# B&R Automation Studio project MotionTestBenchMaster (part 7)

#### FB_ITC.st
```iecst
FUNCTION_BLOCK FB_HMI_ITC_DigitalBool
	VAR_ProgressiveId := INT_TO_UINT(FC_ReminderShift(UINT_TO_INT(Index), 16, 0));

	IF IN_ReadOnly OR IN_HMIAutoForce THEN
		VAR_Auto	:= TRUE;
		VAR_Man		:= FALSE;
	END_IF

	IF IN_IOType THEN
		ITC_IO 	:= SEL(VAR_Auto, VAR_Man, ITC);
	ELSE
		ITC 	:= SEL(VAR_Auto, VAR_Man, ITC_IO);
	END_IF

	IF VAR_OldPage <> HMI_Page.PageNum THEN
		VAR_PageSwitch	:= TRUE;
	END_IF

	IF (Index = (VAR_ProgressiveId + 16 * HMI_Page.PageNum)) AND IN_Visibility THEN
		IF VAR_PageSwitch THEN
			IF IN_IOType THEN
				HMI_Data.DigitalOut[VAR_ProgressiveId].Auto	:= VAR_Auto;
				HMI_Data.DigitalOut[VAR_ProgressiveId].Man	:= VAR_Man;
			ELSE
				HMI_Data.DigitalIn[VAR_ProgressiveId].Auto	:= VAR_Auto;
				HMI_Data.DigitalIn[VAR_ProgressiveId].Man	:= VAR_Man;
			END_IF
			VAR_PageSwitch	:= FALSE;
		END_IF

		IF IN_IOType THEN
			HMI_Data.DigitalOut[VAR_ProgressiveId].Visibility	:= IN_Visibility;
			HMI_Data.DigitalOut[VAR_ProgressiveId].Enable		:= NOT IN_ReadOnly AND NOT IN_HMIAutoForce;
			HMI_Data.DigitalOut[VAR_ProgressiveId].LampState	:= ITC_IO;
			HMI_Data.DigitalOut[VAR_ProgressiveId].Wait			:= IN_Wait;
			HMI_Data.DigitalOut[VAR_ProgressiveId].Alarm		:= IN_Alarm;
			HMI_Data.DigitalOut[VAR_ProgressiveId].Description	:= IN_Description;

			IF EDGEPOS(HMI_Data.DigitalOut[VAR_ProgressiveId].Auto) THEN
				HMI_Data.DigitalOut[VAR_ProgressiveId].Man := FALSE;
			ELSIF EDGEPOS(HMI_Data.DigitalOut[VAR_ProgressiveId].Man) THEN
				HMI_Data.DigitalOut[VAR_ProgressiveId].Auto := FALSE;
			END_IF

			IF IN_ReadOnly OR IN_HMIAutoForce THEN
				HMI_Data.DigitalOut[VAR_ProgressiveId].Auto	:= TRUE;
				HMI_Data.DigitalOut[VAR_ProgressiveId].Man	:= FALSE;
			END_IF

			VAR_Auto	:= HMI_Data.DigitalOut[VAR_ProgressiveId].Auto;
			VAR_Man		:= HMI_Data.DigitalOut[VAR_ProgressiveId].Man;
		ELSE
			HMI_Data.DigitalIn[VAR_ProgressiveId].Visibility	:= IN_Visibility;
			HMI_Data.DigitalIn[VAR_ProgressiveId].Enable		:= NOT IN_ReadOnly AND NOT IN_HMIAutoForce;
			HMI_Data.DigitalIn[VAR_ProgressiveId].LampState 	:= ITC;
			HMI_Data.DigitalIn[VAR_ProgressiveId].Wait			:= IN_Wait;
			HMI_Data.DigitalIn[VAR_ProgressiveId].Alarm			:= IN_Alarm;
			HMI_Data.DigitalIn[VAR_ProgressiveId].Description	:= IN_Description;

			IF EDGEPOS(HMI_Data.DigitalIn[VAR_ProgressiveId].Auto) THEN
				HMI_Data.DigitalIn[VAR_ProgressiveId].Man := FALSE;
			ELSIF EDGEPOS(HMI_Data.DigitalIn[VAR_ProgressiveId].Man) THEN
				HMI_Data.DigitalIn[VAR_ProgressiveId].Auto := FALSE;
			END_IF

			IF IN_ReadOnly OR IN_HMIAutoForce THEN
				HMI_Data.DigitalIn[VAR_ProgressiveId].Auto	:= TRUE;
				HMI_Data.DigitalIn[VAR_ProgressiveId].Man	:= FALSE;
			END_IF

			VAR_Auto	:= HMI_Data.DigitalIn[VAR_ProgressiveId].Auto;
			VAR_Man		:= HMI_Data.DigitalIn[VAR_ProgressiveId].Man;
		END_IF
	ELSIF (Index < (VAR_ProgressiveId + 16 * HMI_Page.PageNum)) THEN
		IF IN_IOType THEN
			HMI_Data.DigitalOut[VAR_ProgressiveId].Visibility	:= FALSE;
		ELSE
			HMI_Data.DigitalIn[VAR_ProgressiveId].Visibility	:= FALSE;
		END_IF
	END_IF

	VAR_OldPage := HMI_Page.PageNum;

	HMI_Data.ManActive	:= NOT VAR_Auto OR HMI_Data.ManActive;

	IF (Index > (16 + 16 * HMI_Page.PageNum)) AND IN_Visibility THEN
		HMI_Data.PageUp.Enable := TRUE;
	END_IF

	IF HMI_Page.PageNum <> 0 THEN
		HMI_Data.PageDown.Enable := TRUE;
	END_IF

	OUT_Man			:= NOT VAR_Auto;
	OUT_ManValue	:= VAR_Man;
	Index			:= Index + 1;
END_FUNCTION_BLOCK

FUNCTION_BLOCK FB_HMI_ITC_DigitalByte
	VAR_ProgressiveId := INT_TO_UINT(FC_ReminderShift(UINT_TO_INT(Index), 16, 0));

	IF IN_ReadOnly OR IN_HMIAutoForce THEN
		VAR_Auto	:= TRUE;
		VAR_Man		:= FALSE;
	END_IF

	IF IN_IOType THEN
		FOR VAR_BitIndex := 0 TO 7 DO
			IF VAR_BitIndex = INT_TO_USINT(IN_BitNumber) THEN
				IF NOT VAR_Auto THEN
					VAR_BitArray[VAR_BitIndex] := VAR_Man;
				ELSE
					VAR_BitArray[VAR_BitIndex] := ITC;
				END_IF
			ELSE
				VAR_BitArray[VAR_BitIndex] := (ITC_IO AND REAL_TO_BYTE(pow(2, VAR_BitIndex))) <> 0;
			END_IF
		END_FOR

		ITC_IO	:= 0;

		FOR VAR_BitIndex := 0 TO 7 DO
			ITC_IO	:= ITC_IO OR UINT_TO_BYTE(((REAL_TO_UINT(pow(2, VAR_BitIndex))) * VAR_BitArray[VAR_BitIndex]));
		END_FOR
	ELSE
		IF NOT VAR_Auto THEN
			ITC		:= VAR_Man;
		ELSE
			ITC		:= (ITC_IO AND REAL_TO_BYTE(pow(2, IN_BitNumber))) <> 0;
		END_IF
	END_IF

	IF VAR_OldPage <> HMI_Page.PageNum THEN
		VAR_PageSwitch	:= TRUE;
	END_IF

	IF (Index = (VAR_ProgressiveId + 16 * HMI_Page.PageNum)) AND IN_Visibility THEN
		IF VAR_PageSwitch THEN
			IF IN_IOType THEN
				HMI_Data.DigitalOut[VAR_ProgressiveId].Auto	:= VAR_Auto;
				HMI_Data.DigitalOut[VAR_ProgressiveId].Man	:= VAR_Man;
			ELSE
				HMI_Data.DigitalIn[VAR_ProgressiveId].Auto	:= VAR_Auto;
				HMI_Data.DigitalIn[VAR_ProgressiveId].Man	:= VAR_Man;
			END_IF
			VAR_PageSwitch	:= FALSE;
		END_IF

		IF IN_IOType THEN
			HMI_Data.DigitalOut[VAR_ProgressiveId].Visibility	:= IN_Visibility;
			HMI_Data.DigitalOut[VAR_ProgressiveId].Enable		:= NOT IN_ReadOnly AND NOT IN_HMIAutoForce;
			HMI_Data.DigitalOut[VAR_ProgressiveId].LampState	:= (ITC_IO AND REAL_TO_BYTE(pow(2, IN_BitNumber))) <> 0;
			HMI_Data.DigitalOut[VAR_ProgressiveId].Wait			:= IN_Wait;
			HMI_Data.DigitalOut[VAR_ProgressiveId].Alarm		:= IN_Alarm;
			HMI_Data.DigitalOut[VAR_ProgressiveId].Description	:= IN_Description;

			IF EDGEPOS(HMI_Data.DigitalOut[VAR_ProgressiveId].Auto) THEN
				HMI_Data.DigitalOut[VAR_ProgressiveId].Man := FALSE;
			ELSIF EDGEPOS(HMI_Data.DigitalOut[VAR_ProgressiveId].Man) THEN
				HMI_Data.DigitalOut[VAR_ProgressiveId].Auto := FALSE;
			END_IF

			IF IN_ReadOnly OR IN_HMIAutoForce THEN
				HMI_Data.DigitalOut[VAR_ProgressiveId].Auto	:= TRUE;
				HMI_Data.DigitalOut[VAR_ProgressiveId].Man	:= FALSE;
			END_IF

			VAR_Auto	:= HMI_Data.DigitalOut[VAR_ProgressiveId].Auto;
			VAR_Man		:= HMI_Data.DigitalOut[VAR_ProgressiveId].Man;
		ELSE
			HMI_Data.DigitalIn[VAR_ProgressiveId].Visibility	:= IN_Visibility;
			HMI_Data.DigitalIn[VAR_ProgressiveId].Enable		:= NOT IN_ReadOnly AND NOT IN_HMIAutoForce;
			HMI_Data.DigitalIn[VAR_ProgressiveId].LampState 	:= ITC;
			HMI_Data.DigitalIn[VAR_ProgressiveId].Wait			:= IN_Wait;
			HMI_Data.DigitalIn[VAR_ProgressiveId].Alarm			:= IN_Alarm;
			HMI_Data.DigitalIn[VAR_ProgressiveId].Description	:= IN_Description;

			IF EDGEPOS(HMI_Data.DigitalIn[VAR_ProgressiveId].Auto) THEN
				HMI_Data.DigitalIn[VAR_ProgressiveId].Man := FALSE;
			ELSIF EDGEPOS(HMI_Data.DigitalIn[VAR_ProgressiveId].Man) THEN
				HMI_Data.DigitalIn[VAR_ProgressiveId].Auto := FALSE;
			END_IF

			IF IN_ReadOnly OR IN_HMIAutoForce THEN
				HMI_Data.DigitalIn[VAR_ProgressiveId].Auto	:= TRUE;
				HMI_Data.DigitalIn[VAR_ProgressiveId].Man	:= FALSE;
			END_IF

			VAR_Auto	:= HMI_Data.DigitalIn[VAR_ProgressiveId].Auto;
			VAR_Man		:= HMI_Data.DigitalIn[VAR_ProgressiveId].Man;
		END_IF
	ELSIF (Index < (VAR_ProgressiveId + 16 * HMI_Page.PageNum)) THEN
		IF IN_IOType THEN
			HMI_Data.DigitalOut[VAR_ProgressiveId].Visibility	:= FALSE;
		ELSE
			HMI_Data.DigitalIn[VAR_ProgressiveId].Visibility	:= FALSE;
		END_IF
	END_IF

	VAR_OldPage := HMI_Page.PageNum;

	HMI_Data.ManActive	:= NOT VAR_Auto OR HMI_Data.ManActive;

	IF (Index > (16 + 16 * HMI_Page.PageNum)) AND IN_Visibility THEN
		HMI_Data.PageUp.Enable := TRUE;
	END_IF

	IF HMI_Page.PageNum <> 0 THEN
		HMI_Data.PageDown.Enable := TRUE;
	END_IF

	OUT_Man			:= NOT VAR_Auto;
	OUT_ManValue	:= VAR_Man;
	Index			:= Index + 1;
END_FUNCTION_BLOCK

FUNCTION_BLOCK FB_HMI_ITC_DigitalUsint
	VAR_ProgressiveId := INT_TO_UINT(FC_ReminderShift(UINT_TO_INT(Index), 16, 0));

	IF IN_ReadOnly OR IN_HMIAutoForce THEN
		VAR_Auto	:= TRUE;
		VAR_Man		:= FALSE;
	END_IF

	IF IN_IOType THEN
		FOR VAR_BitIndex := 0 TO 7 DO
			IF VAR_BitIndex = INT_TO_USINT(IN_BitNumber) THEN
				IF NOT VAR_Auto THEN
					VAR_BitArray[VAR_BitIndex] := VAR_Man;
				ELSE
					VAR_BitArray[VAR_BitIndex] := ITC;
				END_IF
			ELSE
				VAR_BitArray[VAR_BitIndex] := (ITC_IO AND REAL_TO_USINT(pow(2, VAR_BitIndex))) <> 0;
			END_IF
		END_FOR

		ITC_IO	:= 0;

		FOR VAR_BitIndex := 0 TO 7 DO
			ITC_IO	:= ITC_IO OR UINT_TO_USINT(((REAL_TO_UINT(pow(2, VAR_BitIndex))) * VAR_BitArray[VAR_BitIndex]));
		END_FOR
	ELSE
		IF NOT VAR_Auto THEN
			ITC		:= VAR_Man;
		ELSE
			ITC		:= (ITC_IO AND REAL_TO_USINT(pow(2, IN_BitNumber))) <> 0;
		END_IF
	END_IF

	IF VAR_OldPage <> HMI_Page.PageNum THEN
		VAR_PageSwitch	:= TRUE;
	END_IF

	IF (Index = (VAR_ProgressiveId + 16 * HMI_Page.PageNum(*VAR_OldPage*))) AND IN_Visibility THEN
		IF VAR_PageSwitch THEN
			IF IN_IOType THEN
				HMI_Data.DigitalOut[VAR_ProgressiveId].Auto	:= VAR_Auto;
				HMI_Data.DigitalOut[VAR_ProgressiveId].Man	:= VAR_Man;
			ELSE
				HMI_Data.DigitalIn[VAR_ProgressiveId].Auto	:= VAR_Auto;
				HMI_Data.DigitalIn[VAR_ProgressiveId].Man	:= VAR_Man;
			END_IF
			VAR_PageSwitch	:= FALSE;
		END_IF

		IF IN_IOType THEN
			HMI_Data.DigitalOut[VAR_ProgressiveId].Visibility	:= IN_Visibility;
			HMI_Data.DigitalOut[VAR_ProgressiveId].Enable		:= NOT IN_ReadOnly AND NOT IN_HMIAutoForce;
			HMI_Data.DigitalOut[VAR_ProgressiveId].LampState	:= (ITC_IO AND REAL_TO_USINT(pow(2, IN_BitNumber))) <> 0;
			HMI_Data.DigitalOut[VAR_ProgressiveId].Wait			:= IN_Wait;
			HMI_Data.DigitalOut[VAR_ProgressiveId].Alarm		:= IN_Alarm;
			HMI_Data.DigitalOut[VAR_ProgressiveId].Description	:= IN_Description;

			IF EDGEPOS(HMI_Data.DigitalOut[VAR_ProgressiveId].Auto) THEN
				HMI_Data.DigitalOut[VAR_ProgressiveId].Man := FALSE;
				VAR_Man		:= FALSE;
			ELSIF EDGEPOS(HMI_Data.DigitalOut[VAR_ProgressiveId].Man) THEN
				HMI_Data.DigitalOut[VAR_ProgressiveId].Auto := FALSE;
				VAR_Auto	:= FALSE;
			END_IF

			IF IN_ReadOnly OR IN_HMIAutoForce THEN
				HMI_Data.DigitalOut[VAR_ProgressiveId].Auto	:= TRUE;
				HMI_Data.DigitalOut[VAR_ProgressiveId].Man	:= FALSE;
			END_IF

			VAR_Auto	:= HMI_Data.DigitalOut[VAR_ProgressiveId].Auto;
			VAR_Man		:= HMI_Data.DigitalOut[VAR_ProgressiveId].Man;
		ELSE
			HMI_Data.DigitalIn[VAR_ProgressiveId].Visibility	:= IN_Visibility;
			HMI_Data.DigitalIn[VAR_ProgressiveId].Enable		:= NOT IN_ReadOnly AND NOT IN_HMIAutoForce;
			HMI_Data.DigitalIn[VAR_ProgressiveId].LampState 	:= ITC;
			HMI_Data.DigitalIn[VAR_ProgressiveId].Wait			:= IN_Wait;
			HMI_Data.DigitalIn[VAR_ProgressiveId].Alarm			:= IN_Alarm;
			HMI_Data.DigitalIn[VAR_ProgressiveId].Description	:= IN_Description;

			IF EDGEPOS(HMI_Data.DigitalIn[VAR_ProgressiveId].Auto) THEN
				HMI_Data.DigitalIn[VAR_ProgressiveId].Man := FALSE;
			ELSIF EDGEPOS(HMI_Data.DigitalIn[VAR_ProgressiveId].Man) THEN
				HMI_Data.DigitalIn[VAR_ProgressiveId].Auto := FALSE;
			END_IF

			IF IN_ReadOnly OR IN_HMIAutoForce THEN
				HMI_Data.DigitalIn[VAR_ProgressiveId].Auto	:= TRUE;
				HMI_Data.DigitalIn[VAR_ProgressiveId].Man	:= FALSE;
			END_IF

			VAR_Auto	:= HMI_Data.DigitalIn[VAR_ProgressiveId].Auto;
			VAR_Man		:= HMI_Data.DigitalIn[VAR_ProgressiveId].Man;
		END_IF
	ELSIF (Index < (VAR_ProgressiveId + 16 * HMI_Page.PageNum(*VAR_OldPage*))) THEN
		IF IN_IOType THEN
			HMI_Data.DigitalOut[VAR_ProgressiveId].Visibility	:= FALSE;
		ELSE
			HMI_Data.DigitalIn[VAR_ProgressiveId].Visibility	:= FALSE;
		END_IF
	END_IF

	VAR_OldPage := HMI_Page.PageNum;

	HMI_Data.ManActive	:= NOT VAR_Auto OR HMI_Data.ManActive;

	IF (Index > (16 + 16 * HMI_Page.PageNum)) AND IN_Visibility THEN
		HMI_Data.PageUp.Enable := TRUE;
	END_IF

	IF HMI_Page.PageNum <> 0 THEN
		HMI_Data.PageDown.Enable := TRUE;
	END_IF

	OUT_Man			:= NOT VAR_Auto;
	OUT_ManValue	:= VAR_Man;
	Index			:= Index + 1;
END_FUNCTION_BLOCK

FUNCTION_BLOCK FB_HMI_ITC_DigitalInt
	VAR_ProgressiveId := INT_TO_UINT(FC_ReminderShift(UINT_TO_INT(Index), 16, 0));

	IF IN_ReadOnly OR IN_HMIAutoForce THEN
		VAR_Auto	:= TRUE;
		VAR_Man		:= FALSE;
	END_IF

	IF IN_IOType THEN
		FOR VAR_BitIndex := 0 TO 15 DO
			IF VAR_BitIndex = INT_TO_USINT(IN_BitNumber) THEN
				IF NOT VAR_Auto THEN
					VAR_BitArray[VAR_BitIndex] := VAR_Man;
				ELSE
					VAR_BitArray[VAR_BitIndex] := ITC;
				END_IF
			ELSE
				VAR_BitArray[VAR_BitIndex] := (ITC_IO AND REAL_TO_INT(pow(2, VAR_BitIndex))) <> 0;
			END_IF
		END_FOR

		ITC_IO	:= 0;

		FOR VAR_BitIndex := 0 TO 15 DO
			ITC_IO	:= ITC_IO OR UINT_TO_INT(((REAL_TO_UINT(pow(2, VAR_BitIndex))) * VAR_BitArray[VAR_BitIndex]));
		END_FOR
	ELSE
		IF NOT VAR_Auto THEN
			ITC		:= VAR_Man;
		ELSE
			ITC		:= (ITC_IO AND REAL_TO_INT(pow(2, IN_BitNumber))) <> 0;
		END_IF
	END_IF

	IF VAR_OldPage <> HMI_Page.PageNum THEN
		VAR_PageSwitch	:= TRUE;
	END_IF

	IF (Index = (VAR_ProgressiveId + 16 * HMI_Page.PageNum)) AND IN_Visibility THEN
		IF VAR_PageSwitch THEN
			IF IN_IOType THEN
				HMI_Data.DigitalOut[VAR_ProgressiveId].Auto	:= VAR_Auto;
				HMI_Data.DigitalOut[VAR_ProgressiveId].Man	:= VAR_Man;
			ELSE
				HMI_Data.DigitalIn[VAR_ProgressiveId].Auto	:= VAR_Auto;
				HMI_Data.DigitalIn[VAR_ProgressiveId].Man	:= VAR_Man;
			END_IF
			VAR_PageSwitch	:= FALSE;
		END_IF

		IF IN_IOType THEN
			HMI_Data.DigitalOut[VAR_ProgressiveId].Visibility	:= IN_Visibility;
			HMI_Data.DigitalOut[VAR_ProgressiveId].Enable		:= NOT IN_ReadOnly AND NOT IN_HMIAutoForce;
			HMI_Data.DigitalOut[VAR_ProgressiveId].LampState	:= (ITC_IO AND REAL_TO_INT(pow(2, IN_BitNumber))) <> 0;
			HMI_Data.DigitalOut[VAR_ProgressiveId].Wait			:= IN_Wait;
			HMI_Data.DigitalOut[VAR_ProgressiveId].Alarm		:= IN_Alarm;
			HMI_Data.DigitalOut[VAR_ProgressiveId].Description	:= IN_Description;

			IF EDGEPOS(HMI_Data.DigitalOut[VAR_ProgressiveId].Auto) THEN
				HMI_Data.DigitalOut[VAR_ProgressiveId].Man := FALSE;
			ELSIF EDGEPOS(HMI_Data.DigitalOut[VAR_ProgressiveId].Man) THEN
				HMI_Data.DigitalOut[VAR_ProgressiveId].Auto := FALSE;
			END_IF

			VAR_Auto	:= HMI_Data.DigitalOut[VAR_ProgressiveId].Auto;
			VAR_Man		:= HMI_Data.DigitalOut[VAR_ProgressiveId].Man;
		ELSE
			HMI_Data.DigitalIn[VAR_ProgressiveId].Visibility	:= IN_Visibility;
			HMI_Data.DigitalIn[VAR_ProgressiveId].Enable		:= NOT IN_ReadOnly AND NOT IN_HMIAutoForce;
			HMI_Data.DigitalIn[VAR_ProgressiveId].LampState 	:= ITC;
			HMI_Data.DigitalIn[VAR_ProgressiveId].Wait			:= IN_Wait;
			HMI_Data.DigitalIn[VAR_ProgressiveId].Alarm			:= IN_Alarm;
			HMI_Data.DigitalIn[VAR_ProgressiveId].Description	:= IN_Description;

			IF EDGEPOS(HMI_Data.DigitalIn[VAR_ProgressiveId].Auto) THEN
				HMI_Data.DigitalIn[VAR_ProgressiveId].Man := FALSE;
			ELSIF EDGEPOS(HMI_Data.DigitalIn[VAR_ProgressiveId].Man) THEN
				HMI_Data.DigitalIn[VAR_ProgressiveId].Auto := FALSE;
			END_IF

			VAR_Auto	:= HMI_Data.DigitalIn[VAR_ProgressiveId].Auto;
			VAR_Man		:= HMI_Data.DigitalIn[VAR_ProgressiveId].Man;
		END_IF
	ELSIF (Index < (VAR_ProgressiveId + 16 * HMI_Page.PageNum)) THEN
		IF IN_IOType THEN
			HMI_Data.DigitalOut[VAR_ProgressiveId].Visibility	:= FALSE;
		ELSE
			HMI_Data.DigitalIn[VAR_ProgressiveId].Visibility	:= FALSE;
		END_IF
	END_IF

	VAR_OldPage := HMI_Page.PageNum;

	HMI_Data.ManActive	:= NOT VAR_Auto OR HMI_Data.ManActive;

	IF (Index > (16 + 16 * HMI_Page.PageNum)) AND IN_Visibility THEN
		HMI_Data.PageUp.Enable := TRUE;
	END_IF

	IF HMI_Page.PageNum <> 0 THEN
		HMI_Data.PageDown.Enable := TRUE;
	END_IF

	OUT_Man			:= NOT VAR_Auto;
	OUT_ManValue	:= VAR_Man;
	Index			:= Index + 1;
END_FUNCTION_BLOCK

FUNCTION_BLOCK FB_HMI_ITC_AnalogByte
	VAR_ProgressiveId := INT_TO_UINT(FC_ReminderShift(UINT_TO_INT(Index), 4, 0));

	IF IN_ReadOnly OR IN_HMIAutoForce THEN
		VAR_Man		:= FALSE;
	END_IF

	IF IN_IOType THEN
		ITC_IO 		:= SEL(VAR_Man, ITC, VAR_ManValue);
	ELSE
		ITC 		:= SEL(VAR_Man, ITC_IO, VAR_ManValue);
	END_IF

	IF VAR_OldPage <> HMI_Page.PageNum THEN
		VAR_PageSwitch	:= TRUE;
	END_IF

	IF (Index = (VAR_ProgressiveId + 4 * HMI_Page.PageNum)) AND IN_Visibility THEN
		IF VAR_PageSwitch THEN
			IF IN_IOType THEN
				HMI_Data.AnalogOut[VAR_ProgressiveId].Man		:= VAR_Man;
				HMI_Data.AnalogOut[VAR_ProgressiveId].PV_Man	:= BYTE_TO_REAL(VAR_ManValue);
			ELSE
				HMI_Data.AnalogIn[VAR_ProgressiveId].Man		:= VAR_Man;
				HMI_Data.AnalogIn[VAR_ProgressiveId].PV_Man		:= BYTE_TO_REAL(VAR_ManValue);
			END_IF
			VAR_PageSwitch	:= FALSE;
		END_IF

		IF IN_IOType THEN
			HMI_Data.AnalogOut[VAR_ProgressiveId].Visibility	:= IN_Visibility;
			HMI_Data.AnalogOut[VAR_ProgressiveId].Enable		:= NOT IN_ReadOnly AND NOT IN_HMIAutoForce;
			HMI_Data.AnalogOut[VAR_ProgressiveId].PV			:= BYTE_TO_REAL(ITC_IO);
			HMI_Data.AnalogOut[VAR_ProgressiveId].Wait			:= IN_Wait;
			HMI_Data.AnalogOut[VAR_ProgressiveId].Description	:= IN_Description;
			HMI_Data.AnalogOut[VAR_ProgressiveId].Unit			:= IN_Unit;
			HMI_Data.AnalogOut[VAR_ProgressiveId].MaxValue		:= IN_MaxValue;
			HMI_Data.AnalogOut[VAR_ProgressiveId].MinValue		:= IN_MinValue;

			VAR_Man			:= HMI_Data.AnalogOut[VAR_ProgressiveId].Man;
			VAR_ManValue	:= REAL_TO_BYTE(HMI_Data.AnalogOut[VAR_ProgressiveId].PV_Man);
		ELSE
			HMI_Data.AnalogIn[VAR_ProgressiveId].Visibility		:= IN_Visibility;
			HMI_Data.AnalogIn[VAR_ProgressiveId].Enable			:= NOT IN_ReadOnly AND NOT IN_HMIAutoForce;
			HMI_Data.AnalogIn[VAR_ProgressiveId].PV				:= BYTE_TO_REAL(ITC);
			HMI_Data.AnalogIn[VAR_ProgressiveId].Wait			:= IN_Wait;
			HMI_Data.AnalogIn[VAR_ProgressiveId].Description	:= IN_Description;
			HMI_Data.AnalogIn[VAR_ProgressiveId].Unit			:= IN_Unit;
			HMI_Data.AnalogIn[VAR_ProgressiveId].MaxValue		:= IN_MaxValue;
			HMI_Data.AnalogIn[VAR_ProgressiveId].MinValue		:= IN_MinValue;

			VAR_Man			:= HMI_Data.AnalogIn[VAR_ProgressiveId].Man;
			VAR_ManValue	:= REAL_TO_BYTE(HMI_Data.AnalogIn[VAR_ProgressiveId].PV_Man);
		END_IF
	ELSIF (Index < (VAR_ProgressiveId + 4 * HMI_Page.PageNum)) THEN
		IF IN_IOType THEN
			HMI_Data.AnalogOut[VAR_ProgressiveId].Visibility	:= FALSE;
		ELSE
			HMI_Data.AnalogIn[VAR_ProgressiveId].Visibility		:= FALSE;
		END_IF
	END_IF

	VAR_OldPage := HMI_Page.PageNum;

	HMI_Data.ManActive	:= VAR_Man OR HMI_Data.ManActive;

	IF (Index > (4 + 4 * HMI_Page.PageNum)) AND IN_Visibility THEN
		HMI_Data.PageUp.Enable := TRUE;
	END_IF

	IF HMI_Page.PageNum <> 0 THEN
		HMI_Data.PageDown.Enable := TRUE;
	END_IF

	OUT_Man			:= VAR_Man;
	OUT_ManValue	:= VAR_ManValue;
	Index			:= Index + 1;
END_FUNCTION_BLOCK

FUNCTION_BLOCK FB_HMI_ITC_AnalogUsint
	VAR_ProgressiveId := INT_TO_UINT(FC_ReminderShift(UINT_TO_INT(Index), 4, 0));

	IF IN_ReadOnly OR IN_HMIAutoForce THEN
		VAR_Man		:= FALSE;
	END_IF

	IF IN_IOType THEN
		ITC_IO 		:= SEL(VAR_Man, ITC, VAR_ManValue);
	ELSE
		ITC 		:= SEL(VAR_Man, ITC_IO, VAR_ManValue);
	END_IF

	IF VAR_OldPage <> HMI_Page.PageNum THEN
		VAR_PageSwitch	:= TRUE;
	END_IF

	IF (Index = (VAR_ProgressiveId + 4 * HMI_Page.PageNum)) AND IN_Visibility THEN
		IF VAR_PageSwitch THEN
			IF IN_IOType THEN
				HMI_Data.AnalogOut[VAR_ProgressiveId].Man		:= VAR_Man;
				HMI_Data.AnalogOut[VAR_ProgressiveId].PV_Man	:= USINT_TO_REAL(VAR_ManValue);
			ELSE
				HMI_Data.AnalogIn[VAR_ProgressiveId].Man		:= VAR_Man;
				HMI_Data.AnalogIn[VAR_ProgressiveId].PV_Man		:= USINT_TO_REAL(VAR_ManValue);
			END_IF
			VAR_PageSwitch	:= FALSE;
		END_IF

		IF IN_IOType THEN
			HMI_Data.AnalogOut[VAR_ProgressiveId].Visibility	:= IN_Visibility;
			HMI_Data.AnalogOut[VAR_ProgressiveId].Enable		:= NOT IN_ReadOnly AND NOT IN_HMIAutoForce;
			HMI_Data.AnalogOut[VAR_ProgressiveId].PV			:= USINT_TO_REAL(ITC_IO);
			HMI_Data.AnalogOut[VAR_ProgressiveId].Wait			:= IN_Wait;
			HMI_Data.AnalogOut[VAR_ProgressiveId].Description	:= IN_Description;
			HMI_Data.AnalogOut[VAR_ProgressiveId].Unit			:= IN_Unit;
			HMI_Data.AnalogOut[VAR_ProgressiveId].MaxValue		:= IN_MaxValue;
			HMI_Data.AnalogOut[VAR_ProgressiveId].MinValue		:= IN_MinValue;

			VAR_Man			:= HMI_Data.AnalogOut[VAR_ProgressiveId].Man;
			VAR_ManValue	:= REAL_TO_USINT(HMI_Data.AnalogOut[VAR_ProgressiveId].PV_Man);
		ELSE
			HMI_Data.AnalogIn[VAR_ProgressiveId].Visibility		:= IN_Visibility;
			HMI_Data.AnalogIn[VAR_ProgressiveId].Enable			:= NOT IN_ReadOnly AND NOT IN_HMIAutoForce;
			HMI_Data.AnalogIn[VAR_ProgressiveId].PV				:= USINT_TO_REAL(ITC);
			HMI_Data.AnalogIn[VAR_ProgressiveId].Wait			:= IN_Wait;
			HMI_Data.AnalogIn[VAR_ProgressiveId].Description	:= IN_Description;
			HMI_Data.AnalogIn[VAR_ProgressiveId].Unit			:= IN_Unit;
			HMI_Data.AnalogIn[VAR_ProgressiveId].MaxValue		:= IN_MaxValue;
			HMI_Data.AnalogIn[VAR_ProgressiveId].MinValue		:= IN_MinValue;

			VAR_Man			:= HMI_Data.AnalogIn[VAR_ProgressiveId].Man;
			VAR_ManValue	:= REAL_TO_USINT(HMI_Data.AnalogIn[VAR_ProgressiveId].PV_Man);
		END_IF
	ELSIF (Index < (VAR_ProgressiveId + 4 * HMI_Page.PageNum)) THEN
		IF IN_IOType THEN
			HMI_Data.AnalogOut[VAR_ProgressiveId].Visibility	:= FALSE;
		ELSE
			HMI_Data.AnalogIn[VAR_ProgressiveId].Visibility		:= FALSE;
		END_IF
	END_IF

	VAR_OldPage := HMI_Page.PageNum;

	HMI_Data.ManActive	:= VAR_Man OR HMI_Data.ManActive;

	IF (Index > (4 + 4 * HMI_Page.PageNum)) AND IN_Visibility THEN
		HMI_Data.PageUp.Enable := TRUE;
	END_IF

	IF HMI_Page.PageNum <> 0 THEN
		HMI_Data.PageDown.Enable := TRUE;
	END_IF

	OUT_Man			:= VAR_Man;
	OUT_ManValue	:= VAR_ManValue;
	Index			:= Index + 1;
END_FUNCTION_BLOCK

FUNCTION_BLOCK FB_HMI_ITC_AnalogInt
	VAR_ProgressiveId := INT_TO_UINT(FC_ReminderShift(UINT_TO_INT(Index), 4, 0));

	IF IN_ReadOnly OR IN_HMIAutoForce THEN
		VAR_Man		:= FALSE;
	END_IF

	IF IN_IOType THEN
		VAR_Value 	:= SEL(VAR_Man, ITC, VAR_ManValue);
		ITC_IO 		:= SEL(HMI_Data.ComSwap, VAR_Value, swapINT(VAR_Value));
	ELSE
		VAR_Value 	:= SEL(HMI_Data.ComSwap, ITC_IO, swapINT(ITC_IO));
		ITC 		:= SEL(VAR_Man, VAR_Value, VAR_ManValue);
	END_IF

	IF VAR_OldPage <> HMI_Page.PageNum THEN
		VAR_PageSwitch	:= TRUE;
	END_IF

	IF (Index = (VAR_ProgressiveId + 4 * HMI_Page.PageNum)) AND IN_Visibility THEN
		IF VAR_PageSwitch THEN
			IF IN_IOType THEN
				HMI_Data.AnalogOut[VAR_ProgressiveId].Man		:= VAR_Man;
				HMI_Data.AnalogOut[VAR_ProgressiveId].PV_Man	:= INT_TO_REAL(VAR_ManValue);
			ELSE
				HMI_Data.AnalogIn[VAR_ProgressiveId].Man		:= VAR_Man;
				HMI_Data.AnalogIn[VAR_ProgressiveId].PV_Man		:= INT_TO_REAL(VAR_ManValue);
			END_IF
			VAR_PageSwitch	:= FALSE;
		END_IF

		IF IN_IOType THEN
			HMI_Data.AnalogOut[VAR_ProgressiveId].Visibility	:= IN_Visibility;
			HMI_Data.AnalogOut[VAR_ProgressiveId].Enable		:= NOT IN_ReadOnly AND NOT IN_HMIAutoForce;
			HMI_Data.AnalogOut[VAR_ProgressiveId].PV			:= INT_TO_REAL(VAR_Value);
			HMI_Data.AnalogOut[VAR_ProgressiveId].Wait			:= IN_Wait;
			HMI_Data.AnalogOut[VAR_ProgressiveId].Description	:= IN_Description;
			HMI_Data.AnalogOut[VAR_ProgressiveId].Unit			:= IN_Unit;
			HMI_Data.AnalogOut[VAR_ProgressiveId].MaxValue		:= IN_MaxValue;
			HMI_Data.AnalogOut[VAR_ProgressiveId].MinValue		:= IN_MinValue;

			VAR_Man			:= HMI_Data.AnalogOut[VAR_ProgressiveId].Man;
			VAR_ManValue	:= REAL_TO_INT(HMI_Data.AnalogOut[VAR_ProgressiveId].PV_Man);
		ELSE
			HMI_Data.AnalogIn[VAR_ProgressiveId].Visibility		:= IN_Visibility;
			HMI_Data.AnalogIn[VAR_ProgressiveId].Enable			:= NOT IN_ReadOnly AND NOT IN_HMIAutoForce;
			HMI_Data.AnalogIn[VAR_ProgressiveId].PV				:= INT_TO_REAL(ITC);
			HMI_Data.AnalogIn[VAR_ProgressiveId].Wait			:= IN_Wait;
			HMI_Data.AnalogIn[VAR_ProgressiveId].Description	:= IN_Description;
			HMI_Data.AnalogIn[VAR_ProgressiveId].Unit			:= IN_Unit;
			HMI_Data.AnalogIn[VAR_ProgressiveId].MaxValue		:= IN_MaxValue;
			HMI_Data.AnalogIn[VAR_ProgressiveId].MinValue		:= IN_MinValue;

			VAR_Man			:= HMI_Data.AnalogIn[VAR_ProgressiveId].Man;
			VAR_ManValue	:= REAL_TO_INT(HMI_Data.AnalogIn[VAR_ProgressiveId].PV_Man);
		END_IF
	ELSIF (Index < (VAR_ProgressiveId + 4 * HMI_Page.PageNum)) THEN
		IF IN_IOType THEN
			HMI_Data.AnalogOut[VAR_ProgressiveId].Visibility	:= FALSE;
		ELSE
			HMI_Data.AnalogIn[VAR_ProgressiveId].Visibility		:= FALSE;
		END_IF
	END_IF

	VAR_OldPage := HMI_Page.PageNum;

	HMI_Data.ManActive	:= VAR_Man OR HMI_Data.ManActive;

	IF (Index > (4 + 4 * HMI_Page.PageNum)) AND IN_Visibility THEN
		HMI_Data.PageUp.Enable := TRUE;
	END_IF

	IF HMI_Page.PageNum <> 0 THEN
		HMI_Data.PageDown.Enable := TRUE;
	END_IF

	OUT_Man			:= VAR_Man;
	OUT_ManValue	:= VAR_ManValue;
	Index			:= Index + 1;
END_FUNCTION_BLOCK

FUNCTION_BLOCK FB_HMI_ITC_AnalogIntOverUsint
	VAR_ProgressiveId := INT_TO_UINT(FC_ReminderShift(UINT_TO_INT(Index), 4, 0));

	IF IN_ReadOnly OR IN_HMIAutoForce THEN
		VAR_Man		:= FALSE;
	END_IF

	IF IN_IOType THEN
		VAR_Value		:= SEL(VAR_Man, ITC, VAR_ManValue);
		VAR_RawValue	:= SEL(HMI_Data.ComSwap, VAR_Value, swapINT(VAR_Value));
		memcpy(ADR(ITC_IO), ADR(VAR_RawValue), SIZEOF(ITC));
	ELSE
		memcpy(ADR(VAR_RawValue), ADR(ITC_IO), SIZEOF(ITC));
		VAR_Value	:= SEL(HMI_Data.ComSwap, VAR_RawValue, swapINT(VAR_RawValue));
		ITC			:= SEL(VAR_Man, VAR_Value, VAR_ManValue);
	END_IF

	IF VAR_OldPage <> HMI_Page.PageNum THEN
		VAR_PageSwitch	:= TRUE;
	END_IF

	IF (Index = (VAR_ProgressiveId + 4 * HMI_Page.PageNum)) AND IN_Visibility THEN
		IF VAR_PageSwitch THEN
			IF IN_IOType THEN
				HMI_Data.AnalogOut[VAR_ProgressiveId].Man		:= VAR_Man;
				HMI_Data.AnalogOut[VAR_ProgressiveId].PV_Man	:= INT_TO_REAL(VAR_ManValue);
			ELSE
				HMI_Data.AnalogIn[VAR_ProgressiveId].Man		:= VAR_Man;
				HMI_Data.AnalogIn[VAR_ProgressiveId].PV_Man		:= INT_TO_REAL(VAR_ManValue);
			END_IF
			VAR_PageSwitch	:= FALSE;
		END_IF

		IF IN_IOType THEN
			HMI_Data.AnalogOut[VAR_ProgressiveId].Visibility	:= IN_Visibility;
			HMI_Data.AnalogOut[VAR_ProgressiveId].Enable		:= NOT IN_ReadOnly AND NOT IN_HMIAutoForce;
			HMI_Data.AnalogOut[VAR_ProgressiveId].PV			:= INT_TO_REAL(VAR_Value);
			HMI_Data.AnalogOut[VAR_ProgressiveId].Wait			:= IN_Wait;
			HMI_Data.AnalogOut[VAR_ProgressiveId].Description	:= IN_Description;
			HMI_Data.AnalogOut[VAR_ProgressiveId].Unit			:= IN_Unit;
			HMI_Data.AnalogOut[VAR_ProgressiveId].MaxValue		:= IN_MaxValue;
			HMI_Data.AnalogOut[VAR_ProgressiveId].MinValue		:= IN_MinValue;

			VAR_Man			:= HMI_Data.AnalogOut[VAR_ProgressiveId].Man;
			VAR_ManValue	:= REAL_TO_INT(HMI_Data.AnalogOut[VAR_ProgressiveId].PV_Man);
		ELSE
			HMI_Data.AnalogIn[VAR_ProgressiveId].Visibility		:= IN_Visibility;
			HMI_Data.AnalogIn[VAR_ProgressiveId].Enable			:= NOT IN_ReadOnly AND NOT IN_HMIAutoForce;
			HMI_Data.AnalogIn[VAR_ProgressiveId].PV				:= INT_TO_REAL(ITC);
			HMI_Data.AnalogIn[VAR_ProgressiveId].Wait			:= IN_Wait;
			HMI_Data.AnalogIn[VAR_ProgressiveId].Description	:= IN_Description;
			HMI_Data.AnalogIn[VAR_ProgressiveId].Unit			:= IN_Unit;
			HMI_Data.AnalogIn[VAR_ProgressiveId].MaxValue		:= IN_MaxValue;
			HMI_Data.AnalogIn[VAR_ProgressiveId].MinValue		:= IN_MinValue;

			VAR_Man			:= HMI_Data.AnalogIn[VAR_ProgressiveId].Man;
			VAR_ManValue	:= REAL_TO_INT(HMI_Data.AnalogIn[VAR_ProgressiveId].PV_Man);
		END_IF
	ELSIF (Index < (VAR_ProgressiveId + 4 * HMI_Page.PageNum)) THEN
		IF IN_IOType THEN
			HMI_Data.AnalogOut[VAR_ProgressiveId].Visibility	:= FALSE;
		ELSE
			HMI_Data.AnalogIn[VAR_ProgressiveId].Visibility		:= FALSE;
		END_IF
	END_IF

	VAR_OldPage := HMI_Page.PageNum;

	HMI_Data.ManActive	:= VAR_Man OR HMI_Data.ManActive;

	IF (Index > (4 + 4 * HMI_Page.PageNum)) AND IN_Visibility THEN
		HMI_Data.PageUp.Enable := TRUE;
	END_IF

	IF HMI_Page.PageNum <> 0 THEN
		HMI_Data.PageDown.Enable := TRUE;
	END_IF

	OUT_Man			:= VAR_Man;
	OUT_ManValue	:= VAR_ManValue;
	Index			:= Index + 1;
END_FUNCTION_BLOCK

FUNCTION_BLOCK FB_HMI_ITC_AnalogUintOverUsint
	VAR_ProgressiveId := INT_TO_UINT(FC_ReminderShift(UINT_TO_INT(Index), 4, 0));

	IF IN_ReadOnly OR IN_HMIAutoForce THEN
		VAR_Man		:= FALSE;
	END_IF

	IF IN_IOType THEN
		VAR_Value		:= SEL(VAR_Man, ITC, VAR_ManValue);
		VAR_RawValue	:= SEL(HMI_Data.ComSwap, VAR_Value, swapINT(VAR_Value));
		memcpy(ADR(ITC_IO), ADR(VAR_RawValue), SIZEOF(ITC));
	ELSE
		memcpy(ADR(VAR_RawValue), ADR(ITC_IO), SIZEOF(ITC));
		VAR_Value	:= SEL(HMI_Data.ComSwap, VAR_RawValue, swapINT(VAR_RawValue));
		ITC			:= SEL(VAR_Man, VAR_Value, VAR_ManValue);
	END_IF

	IF VAR_OldPage <> HMI_Page.PageNum THEN
		VAR_PageSwitch	:= TRUE;
	END_IF

	IF (Index = (VAR_ProgressiveId + 4 * HMI_Page.PageNum)) AND IN_Visibility THEN
		IF VAR_PageSwitch THEN
			IF IN_IOType THEN
				HMI_Data.AnalogOut[VAR_ProgressiveId].Man		:= VAR_Man;
				HMI_Data.AnalogOut[VAR_ProgressiveId].PV_Man	:= INT_TO_REAL(VAR_ManValue);
			ELSE
				HMI_Data.AnalogIn[VAR_ProgressiveId].Man		:= VAR_Man;
				HMI_Data.AnalogIn[VAR_ProgressiveId].PV_Man		:= INT_TO_REAL(VAR_ManValue);
			END_IF
			VAR_PageSwitch	:= FALSE;
		END_IF

		IF IN_IOType THEN
			HMI_Data.AnalogOut[VAR_ProgressiveId].Visibility	:= IN_Visibility;
			HMI_Data.AnalogOut[VAR_ProgressiveId].Enable		:= NOT IN_ReadOnly AND NOT IN_HMIAutoForce;
			HMI_Data.AnalogOut[VAR_ProgressiveId].PV			:= INT_TO_REAL(VAR_Value);
			HMI_Data.AnalogOut[VAR_ProgressiveId].Wait			:= IN_Wait;
			HMI_Data.AnalogOut[VAR_ProgressiveId].Description	:= IN_Description;
			HMI_Data.AnalogOut[VAR_ProgressiveId].Unit			:= IN_Unit;
			HMI_Data.AnalogOut[VAR_ProgressiveId].MaxValue		:= IN_MaxValue;
			HMI_Data.AnalogOut[VAR_ProgressiveId].MinValue		:= IN_MinValue;

			VAR_Man			:= HMI_Data.AnalogOut[VAR_ProgressiveId].Man;
			VAR_ManValue	:= REAL_TO_INT(HMI_Data.AnalogOut[VAR_ProgressiveId].PV_Man);
		ELSE
			HMI_Data.AnalogIn[VAR_ProgressiveId].Visibility		:= IN_Visibility;
			HMI_Data.AnalogIn[VAR_ProgressiveId].Enable			:= NOT IN_ReadOnly AND NOT IN_HMIAutoForce;
			HMI_Data.AnalogIn[VAR_ProgressiveId].PV				:= INT_TO_REAL(ITC);
			HMI_Data.AnalogIn[VAR_ProgressiveId].Wait			:= IN_Wait;
			HMI_Data.AnalogIn[VAR_ProgressiveId].Description	:= IN_Description;
			HMI_Data.AnalogIn[VAR_ProgressiveId].Unit			:= IN_Unit;
			HMI_Data.AnalogIn[VAR_ProgressiveId].MaxValue		:= IN_MaxValue;
			HMI_Data.AnalogIn[VAR_ProgressiveId].MinValue		:= IN_MinValue;

			VAR_Man			:= HMI_Data.AnalogIn[VAR_ProgressiveId].Man;
			VAR_ManValue	:= REAL_TO_INT(HMI_Data.AnalogIn[VAR_ProgressiveId].PV_Man);
		END_IF
	ELSIF (Index < (VAR_ProgressiveId + 4 * HMI_Page.PageNum)) THEN
		IF IN_IOType THEN
			HMI_Data.AnalogOut[VAR_ProgressiveId].Visibility	:= FALSE;
		ELSE
			HMI_Data.AnalogIn[VAR_ProgressiveId].Visibility		:= FALSE;
		END_IF
	END_IF

	VAR_OldPage := HMI_Page.PageNum;

	HMI_Data.ManActive	:= VAR_Man OR HMI_Data.ManActive;

	IF (Index > (4 + 4 * HMI_Page.PageNum)) AND IN_Visibility THEN
		HMI_Data.PageUp.Enable := TRUE;
	END_IF

	IF HMI_Page.PageNum <> 0 THEN
		HMI_Data.PageDown.Enable := TRUE;
	END_IF

	OUT_Man			:= VAR_Man;
	OUT_ManValue	:= VAR_ManValue;
	Index			:= Index + 1;
END_FUNCTION_BLOCK

FUNCTION_BLOCK FB_HMI_ITC_AnalogDInt
	VAR_ProgressiveId := INT_TO_UINT(FC_ReminderShift(UINT_TO_INT(Index), 4, 0));

	IF IN_ReadOnly OR IN_HMIAutoForce THEN
		VAR_Man		:= FALSE;
	END_IF

	IF IN_IOType THEN
		VAR_Value	:= SEL(VAR_Man, ITC, VAR_ManValue);
		ITC_IO		:= SEL(HMI_Data.ComSwap, VAR_Value, swapDINT(VAR_Value));
	ELSE
		VAR_Value	:= SEL(HMI_Data.ComSwap, ITC_IO, swapDINT(ITC_IO));
		ITC			:= SEL(VAR_Man, VAR_Value, VAR_ManValue);
	END_IF

	IF VAR_OldPage <> HMI_Page.PageNum THEN
		VAR_PageSwitch	:= TRUE;
	END_IF

	IF (Index = (VAR_ProgressiveId + 4 * HMI_Page.PageNum)) AND IN_Visibility THEN
		IF VAR_PageSwitch THEN
			IF IN_IOType THEN
				HMI_Data.AnalogOut[VAR_ProgressiveId].Man		:= VAR_Man;
				HMI_Data.AnalogOut[VAR_ProgressiveId].PV_Man	:= DINT_TO_REAL(VAR_ManValue);
			ELSE
				HMI_Data.AnalogIn[VAR_ProgressiveId].Man		:= VAR_Man;
				HMI_Data.AnalogIn[VAR_ProgressiveId].PV_Man		:= DINT_TO_REAL(VAR_ManValue);
			END_IF
			VAR_PageSwitch	:= FALSE;
		END_IF

		IF IN_IOType THEN
			HMI_Data.AnalogOut[VAR_ProgressiveId].Visibility	:= IN_Visibility;
			HMI_Data.AnalogOut[VAR_ProgressiveId].Enable		:= NOT IN_ReadOnly AND NOT IN_HMIAutoForce;
			HMI_Data.AnalogOut[VAR_ProgressiveId].PV			:= DINT_TO_REAL(VAR_Value);
			HMI_Data.AnalogOut[VAR_ProgressiveId].Wait			:= IN_Wait;
			HMI_Data.AnalogOut[VAR_ProgressiveId].Description	:= IN_Description;
			HMI_Data.AnalogOut[VAR_ProgressiveId].Unit			:= IN_Unit;
			HMI_Data.AnalogOut[VAR_ProgressiveId].MaxValue		:= IN_MaxValue;
			HMI_Data.AnalogOut[VAR_ProgressiveId].MinValue		:= IN_MinValue;

			VAR_Man			:= HMI_Data.AnalogOut[VAR_ProgressiveId].Man;
			VAR_ManValue	:= REAL_TO_INT(HMI_Data.AnalogOut[VAR_ProgressiveId].PV_Man);
		ELSE
			HMI_Data.AnalogIn[VAR_ProgressiveId].Visibility		:= IN_Visibility;
			HMI_Data.AnalogIn[VAR_ProgressiveId].Enable			:= NOT IN_ReadOnly AND NOT IN_HMIAutoForce;
			HMI_Data.AnalogIn[VAR_ProgressiveId].PV				:= DINT_TO_REAL(ITC);
			HMI_Data.AnalogIn[VAR_ProgressiveId].Wait			:= IN_Wait;
			HMI_Data.AnalogIn[VAR_ProgressiveId].Description	:= IN_Description;
			HMI_Data.AnalogIn[VAR_ProgressiveId].Unit			:= IN_Unit;
			HMI_Data.AnalogIn[VAR_ProgressiveId].MaxValue		:= IN_MaxValue;
			HMI_Data.AnalogIn[VAR_ProgressiveId].MinValue		:= IN_MinValue;

			VAR_Man			:= HMI_Data.AnalogIn[VAR_ProgressiveId].Man;
			VAR_ManValue	:= REAL_TO_INT(HMI_Data.AnalogIn[VAR_ProgressiveId].PV_Man);
		END_IF
	ELSIF (Index < (VAR_ProgressiveId + 4 * HMI_Page.PageNum)) THEN
		IF IN_IOType THEN
			HMI_Data.AnalogOut[VAR_ProgressiveId].Visibility	:= FALSE;
		ELSE
			HMI_Data.AnalogIn[VAR_ProgressiveId].Visibility		:= FALSE;
		END_IF
	END_IF

	VAR_OldPage := HMI_Page.PageNum;

	HMI_Data.ManActive	:= VAR_Man OR HMI_Data.ManActive;

	IF (Index > (4 + 4 * HMI_Page.PageNum)) AND IN_Visibility THEN
		HMI_Data.PageUp.Enable := TRUE;
	END_IF

	IF HMI_Page.PageNum <> 0 THEN
		HMI_Data.PageDown.Enable := TRUE;
	END_IF

	OUT_Man			:= VAR_Man;
	OUT_ManValue	:= VAR_ManValue;
	Index	:= Index + 1;
END_FUNCTION_BLOCK

FUNCTION_BLOCK FB_HMI_ITC_AnalogUdint
	VAR_ProgressiveId := INT_TO_UINT(FC_ReminderShift(UINT_TO_INT(Index), 4, 0));

	IF IN_ReadOnly OR IN_HMIAutoForce THEN
		VAR_Man		:= FALSE;
	END_IF

	IF IN_IOType THEN
		VAR_Value	:= SEL(VAR_Man, ITC, VAR_ManValue);
		ITC_IO		:= SEL(HMI_Data.ComSwap, VAR_Value, swapUDINT(VAR_Value));
	ELSE
		VAR_Value	:= SEL(HMI_Data.ComSwap, ITC_IO, swapUDINT(ITC_IO));
		ITC			:= SEL(VAR_Man, VAR_Value, VAR_ManValue);
	END_IF

	IF VAR_OldPage <> HMI_Page.PageNum THEN
		VAR_PageSwitch	:= TRUE;
	END_IF

	IF (Index = (VAR_ProgressiveId + 4 * HMI_Page.PageNum)) AND IN_Visibility THEN
		IF VAR_PageSwitch THEN
			IF IN_IOType THEN
				HMI_Data.AnalogOut[VAR_ProgressiveId].Man		:= VAR_Man;
				HMI_Data.AnalogOut[VAR_ProgressiveId].PV_Man	:= UDINT_TO_REAL(VAR_ManValue);
			ELSE
				HMI_Data.AnalogIn[VAR_ProgressiveId].Man		:= VAR_Man;
				HMI_Data.AnalogIn[VAR_ProgressiveId].PV_Man		:= UDINT_TO_REAL(VAR_ManValue);
			END_IF
			VAR_PageSwitch	:= FALSE;
		END_IF

		IF IN_IOType THEN
			HMI_Data.AnalogOut[VAR_ProgressiveId].Visibility	:= IN_Visibility;
			HMI_Data.AnalogOut[VAR_ProgressiveId].Enable		:= NOT IN_ReadOnly AND NOT IN_HMIAutoForce;
			HMI_Data.AnalogOut[VAR_ProgressiveId].PV			:= UDINT_TO_REAL(VAR_Value);
			HMI_Data.AnalogOut[VAR_ProgressiveId].Wait			:= IN_Wait;
			HMI_Data.AnalogOut[VAR_ProgressiveId].Description	:= IN_Description;
			HMI_Data.AnalogOut[VAR_ProgressiveId].Unit			:= IN_Unit;
			HMI_Data.AnalogOut[VAR_ProgressiveId].MaxValue		:= IN_MaxValue;
			HMI_Data.AnalogOut[VAR_ProgressiveId].MinValue		:= IN_MinValue;

			VAR_Man			:= HMI_Data.AnalogOut[VAR_ProgressiveId].Man;
			VAR_ManValue	:= REAL_TO_INT(HMI_Data.AnalogOut[VAR_ProgressiveId].PV_Man);
		ELSE
			HMI_Data.AnalogIn[VAR_ProgressiveId].Visibility		:= IN_Visibility;
			HMI_Data.AnalogIn[VAR_ProgressiveId].Enable			:= NOT IN_ReadOnly AND NOT IN_HMIAutoForce;
			HMI_Data.AnalogIn[VAR_ProgressiveId].PV				:= UDINT_TO_REAL(ITC);
			HMI_Data.AnalogIn[VAR_ProgressiveId].Wait			:= IN_Wait;
			HMI_Data.AnalogIn[VAR_ProgressiveId].Description	:= IN_Description;
			HMI_Data.AnalogIn[VAR_ProgressiveId].Unit			:= IN_Unit;
			HMI_Data.AnalogIn[VAR_ProgressiveId].MaxValue		:= IN_MaxValue;
			HMI_Data.AnalogIn[VAR_ProgressiveId].MinValue		:= IN_MinValue;

			VAR_Man			:= HMI_Data.AnalogIn[VAR_ProgressiveId].Man;
			VAR_ManValue	:= REAL_TO_INT(HMI_Data.AnalogIn[VAR_ProgressiveId].PV_Man);
		END_IF
	ELSIF (Index < (VAR_ProgressiveId + 4 * HMI_Page.PageNum)) THEN
		IF IN_IOType THEN
			HMI_Data.AnalogOut[VAR_ProgressiveId].Visibility	:= FALSE;
		ELSE
			HMI_Data.AnalogIn[VAR_ProgressiveId].Visibility		:= FALSE;
		END_IF
	END_IF

	VAR_OldPage := HMI_Page.PageNum;

	HMI_Data.ManActive	:= VAR_Man OR HMI_Data.ManActive;

	IF (Index > (4 + 4 * HMI_Page.PageNum)) AND IN_Visibility THEN
		HMI_Data.PageUp.Enable := TRUE;
	END_IF

	IF HMI_Page.PageNum <> 0 THEN
		HMI_Data.PageDown.Enable := TRUE;
	END_IF

	OUT_Man			:= VAR_Man;
	OUT_ManValue	:= VAR_ManValue;
	Index	:= Index + 1;
END_FUNCTION_BLOCK

FUNCTION_BLOCK FB_HMI_ITC_AnalogDIntOverUsint
	VAR_ProgressiveId := INT_TO_UINT(FC_ReminderShift(UINT_TO_INT(Index), 4, 0));

	IF IN_ReadOnly OR IN_HMIAutoForce THEN
		VAR_Man		:= FALSE;
	END_IF

	IF IN_IOType THEN
		VAR_Value		:= SEL(VAR_Man, ITC, VAR_ManValue);
		VAR_RawValue	:= SEL(HMI_Data.ComSwap, VAR_Value, swapDINT(VAR_Value));
		memcpy(ADR(ITC_IO), ADR(VAR_RawValue), SIZEOF(ITC));
	ELSE
		memcpy(ADR(VAR_RawValue), ADR(ITC_IO), SIZEOF(ITC));
		VAR_Value	:= SEL(HMI_Data.ComSwap, VAR_RawValue, swapDINT(VAR_RawValue));
		ITC			:= SEL(VAR_Man, VAR_Value, VAR_ManValue);
	END_IF

	IF VAR_OldPage <> HMI_Page.PageNum THEN
		VAR_PageSwitch	:= TRUE;
	END_IF

	IF (Index = (VAR_ProgressiveId + 4 * HMI_Page.PageNum)) AND IN_Visibility THEN
		IF VAR_PageSwitch THEN
			IF IN_IOType THEN
				HMI_Data.AnalogOut[VAR_ProgressiveId].Man		:= VAR_Man;
				HMI_Data.AnalogOut[VAR_ProgressiveId].PV_Man	:= DINT_TO_REAL(VAR_ManValue);
			ELSE
				HMI_Data.AnalogIn[VAR_ProgressiveId].Man		:= VAR_Man;
				HMI_Data.AnalogIn[VAR_ProgressiveId].PV_Man		:= DINT_TO_REAL(VAR_ManValue);
			END_IF
			VAR_PageSwitch	:= FALSE;
		END_IF

		IF IN_IOType THEN
			HMI_Data.AnalogOut[VAR_ProgressiveId].Visibility	:= IN_Visibility;
			HMI_Data.AnalogOut[VAR_ProgressiveId].Enable		:= NOT IN_ReadOnly AND NOT IN_HMIAutoForce;
			HMI_Data.AnalogOut[VAR_ProgressiveId].PV			:= DINT_TO_REAL(VAR_Value);
			HMI_Data.AnalogOut[VAR_ProgressiveId].Wait			:= IN_Wait;
			HMI_Data.AnalogOut[VAR_ProgressiveId].Description	:= IN_Description;
			HMI_Data.AnalogOut[VAR_ProgressiveId].Unit			:= IN_Unit;
			HMI_Data.AnalogOut[VAR_ProgressiveId].MaxValue		:= IN_MaxValue;
			HMI_Data.AnalogOut[VAR_ProgressiveId].MinValue		:= IN_MinValue;

			VAR_Man			:= HMI_Data.AnalogOut[VAR_ProgressiveId].Man;
			VAR_ManValue	:= REAL_TO_INT(HMI_Data.AnalogOut[VAR_ProgressiveId].PV_Man);
		ELSE
			HMI_Data.AnalogIn[VAR_ProgressiveId].Visibility		:= IN_Visibility;
			HMI_Data.AnalogIn[VAR_ProgressiveId].Enable			:= NOT IN_ReadOnly AND NOT IN_HMIAutoForce;
			HMI_Data.AnalogIn[VAR_ProgressiveId].PV				:= DINT_TO_REAL(ITC);
			HMI_Data.AnalogIn[VAR_ProgressiveId].Wait			:= IN_Wait;
			HMI_Data.AnalogIn[VAR_ProgressiveId].Description	:= IN_Description;
			HMI_Data.AnalogIn[VAR_ProgressiveId].Unit			:= IN_Unit;
			HMI_Data.AnalogIn[VAR_ProgressiveId].MaxValue		:= IN_MaxValue;
			HMI_Data.AnalogIn[VAR_ProgressiveId].MinValue		:= IN_MinValue;

			VAR_Man			:= HMI_Data.AnalogIn[VAR_ProgressiveId].Man;
			VAR_ManValue	:= REAL_TO_INT(HMI_Data.AnalogIn[VAR_ProgressiveId].PV_Man);
		END_IF
	ELSIF (Index < (VAR_ProgressiveId + 4 * HMI_Page.PageNum)) THEN
		IF IN_IOType THEN
			HMI_Data.AnalogOut[VAR_ProgressiveId].Visibility	:= FALSE;
		ELSE
			HMI_Data.AnalogIn[VAR_ProgressiveId].Visibility		:= FALSE;
		END_IF
	END_IF

	VAR_OldPage := HMI_Page.PageNum;

	HMI_Data.ManActive	:= VAR_Man OR HMI_Data.ManActive;

	IF (Index > (4 + 4 * HMI_Page.PageNum)) AND IN_Visibility THEN
		HMI_Data.PageUp.Enable := TRUE;
	END_IF

	IF HMI_Page.PageNum <> 0 THEN
		HMI_Data.PageDown.Enable := TRUE;
	END_IF

	OUT_Man			:= VAR_Man;
	OUT_ManValue	:= VAR_ManValue;
	Index			:= Index + 1;
END_FUNCTION_BLOCK

FUNCTION_BLOCK FB_HMI_ITC_AnalogReal
	VAR_ProgressiveId := INT_TO_UINT(FC_ReminderShift(UINT_TO_INT(Index), 4, 0));

	IF IN_ReadOnly OR IN_HMIAutoForce THEN
		VAR_Man		:= FALSE;
	END_IF

	IF IN_IOType THEN
		VAR_Value	:= SEL(VAR_Man, ITC, VAR_ManValue);
		ITC_IO		:= SEL(HMI_Data.ComSwap, VAR_Value, swapREAL(VAR_Value));
	ELSE
		VAR_Value	:= SEL(HMI_Data.ComSwap, ITC_IO, swapREAL(ITC_IO));
		ITC			:= SEL(VAR_Man, VAR_Value, VAR_ManValue);
	END_IF

	IF VAR_OldPage <> HMI_Page.PageNum THEN
		VAR_PageSwitch	:= TRUE;
	END_IF

	IF (Index = (VAR_ProgressiveId + 4 * HMI_Page.PageNum)) AND IN_Visibility THEN
		IF VAR_PageSwitch THEN
			IF IN_IOType THEN
				HMI_Data.AnalogOut[VAR_ProgressiveId].Man		:= VAR_Man;
				HMI_Data.AnalogOut[VAR_ProgressiveId].PV_Man	:= VAR_ManValue;
			ELSE
				HMI_Data.AnalogIn[VAR_ProgressiveId].Man	:= VAR_Man;
				HMI_Data.AnalogIn[VAR_ProgressiveId].PV_Man	:= VAR_ManValue;
			END_IF
			VAR_PageSwitch	:= FALSE;
		END_IF

		IF IN_IOType THEN
			HMI_Data.AnalogOut[VAR_ProgressiveId].Visibility	:= IN_Visibility;
			HMI_Data.AnalogOut[VAR_ProgressiveId].Enable		:= NOT IN_ReadOnly AND NOT IN_HMIAutoForce;
			HMI_Data.AnalogOut[VAR_ProgressiveId].PV			:= VAR_Value;
			HMI_Data.AnalogOut[VAR_ProgressiveId].Wait			:= IN_Wait;
			HMI_Data.AnalogOut[VAR_ProgressiveId].Description	:= IN_Description;
			HMI_Data.AnalogOut[VAR_ProgressiveId].Unit			:= IN_Unit;
			HMI_Data.AnalogOut[VAR_ProgressiveId].MaxValue		:= IN_MaxValue;
			HMI_Data.AnalogOut[VAR_ProgressiveId].MinValue		:= IN_MinValue;

			VAR_Man			:= HMI_Data.AnalogOut[VAR_ProgressiveId].Man;
			VAR_ManValue	:= HMI_Data.AnalogOut[VAR_ProgressiveId].PV_Man;
		ELSE
			HMI_Data.AnalogIn[VAR_ProgressiveId].Visibility		:= IN_Visibility;
			HMI_Data.AnalogIn[VAR_ProgressiveId].Enable			:= NOT IN_ReadOnly AND NOT IN_HMIAutoForce;
			HMI_Data.AnalogIn[VAR_ProgressiveId].PV				:= ITC;
			HMI_Data.AnalogIn[VAR_ProgressiveId].Wait			:= IN_Wait;
			HMI_Data.AnalogIn[VAR_ProgressiveId].Description	:= IN_Description;
			HMI_Data.AnalogIn[VAR_ProgressiveId].Unit			:= IN_Unit;
			HMI_Data.AnalogIn[VAR_ProgressiveId].MaxValue		:= IN_MaxValue;
			HMI_Data.AnalogIn[VAR_ProgressiveId].MinValue		:= IN_MinValue;

			VAR_Man			:= HMI_Data.AnalogIn[VAR_ProgressiveId].Man;
			VAR_ManValue	:= HMI_Data.AnalogIn[VAR_ProgressiveId].PV_Man;
		END_IF
	ELSIF (Index < (VAR_ProgressiveId + 4 * HMI_Page.PageNum)) THEN
		IF IN_IOType THEN
			HMI_Data.AnalogOut[VAR_ProgressiveId].Visibility	:= FALSE;
		ELSE
			HMI_Data.AnalogIn[VAR_ProgressiveId].Visibility		:= FALSE;
		END_IF
	END_IF

	VAR_OldPage := HMI_Page.PageNum;

	HMI_Data.ManActive	:= VAR_Man OR HMI_Data.ManActive;

	IF (Index > (4 + 4 * HMI_Page.PageNum)) AND IN_Visibility THEN
		HMI_Data.PageUp.Enable := TRUE;
	END_IF

	IF HMI_Page.PageNum <> 0 THEN
		HMI_Data.PageDown.Enable := TRUE;
	END_IF

	OUT_Man			:= VAR_Man;
	OUT_ManValue	:= VAR_ManValue;
	Index			:= Index + 1;
END_FUNCTION_BLOCK

FUNCTION_BLOCK FB_HMI_ITC_AnalogRealOverUsint
	VAR_ProgressiveId := INT_TO_UINT(FC_ReminderShift(UINT_TO_INT(Index), 4, 0));

	IF IN_ReadOnly OR IN_HMIAutoForce THEN
		VAR_Man		:= FALSE;
	END_IF

	IF IN_IOType THEN
		VAR_Value	:= SEL(VAR_Man, ITC, VAR_ManValue);
		VAR_RawValue	:= SEL(HMI_Data.ComSwap, VAR_Value, swapREAL(VAR_Value));
		memcpy(ADR(ITC_IO), ADR(VAR_RawValue), SIZEOF(ITC));
	ELSE
		memcpy(ADR(VAR_RawValue), ADR(ITC_IO), SIZEOF(ITC));
		VAR_Value	:= SEL(HMI_Data.ComSwap, VAR_RawValue, swapREAL(VAR_RawValue));
		ITC		:= SEL(VAR_Man, VAR_Value, VAR_ManValue);
	END_IF

	IF VAR_OldPage <> HMI_Page.PageNum THEN
		VAR_PageSwitch	:= TRUE;
	END_IF

	IF (Index = (VAR_ProgressiveId + 4 * HMI_Page.PageNum)) AND IN_Visibility THEN
		IF VAR_PageSwitch THEN
			IF IN_IOType THEN
				HMI_Data.AnalogOut[VAR_ProgressiveId].Man		:= VAR_Man;
				HMI_Data.AnalogOut[VAR_ProgressiveId].PV_Man	:= VAR_ManValue;
			ELSE
				HMI_Data.AnalogIn[VAR_ProgressiveId].Man		:= VAR_Man;
				HMI_Data.AnalogIn[VAR_ProgressiveId].PV_Man		:= VAR_ManValue;
			END_IF
			VAR_PageSwitch	:= FALSE;
		END_IF

		IF IN_IOType THEN
			HMI_Data.AnalogOut[VAR_ProgressiveId].Visibility	:= IN_Visibility;
			HMI_Data.AnalogOut[VAR_ProgressiveId].Enable		:= NOT IN_ReadOnly AND NOT IN_HMIAutoForce;
			VAR_Value	:= swapREAL(ITC_IO);
			memcpy(ADR(RealValue), ADR(VAR_Value), SIZEOF(RealValue));
			HMI_Data.AnalogOut[VAR_ProgressiveId].PV			:= VAR_Value;
			HMI_Data.AnalogOut[VAR_ProgressiveId].Wait			:= IN_Wait;
			HMI_Data.AnalogOut[VAR_ProgressiveId].Description	:= IN_Description;
			HMI_Data.AnalogOut[VAR_ProgressiveId].Unit			:= IN_Unit;
			HMI_Data.AnalogOut[VAR_ProgressiveId].MaxValue		:= IN_MaxValue;
			HMI_Data.AnalogOut[VAR_ProgressiveId].MinValue		:= IN_MinValue;

			VAR_Man			:= HMI_Data.AnalogOut[VAR_ProgressiveId].Man;
			VAR_ManValue	:= HMI_Data.AnalogOut[VAR_ProgressiveId].PV_Man;
		ELSE
			HMI_Data.AnalogIn[VAR_ProgressiveId].Visibility		:= IN_Visibility;
			HMI_Data.AnalogIn[VAR_ProgressiveId].Enable			:= NOT IN_ReadOnly AND NOT IN_HMIAutoForce;
			HMI_Data.AnalogIn[VAR_ProgressiveId].PV				:= ITC;
			HMI_Data.AnalogIn[VAR_ProgressiveId].Wait			:= IN_Wait;
			HMI_Data.AnalogIn[VAR_ProgressiveId].Description	:= IN_Description;
			HMI_Data.AnalogIn[VAR_ProgressiveId].Unit			:= IN_Unit;
			HMI_Data.AnalogIn[VAR_ProgressiveId].MaxValue		:= IN_MaxValue;
			HMI_Data.AnalogIn[VAR_ProgressiveId].MinValue		:= IN_MinValue;

			VAR_Man			:= HMI_Data.AnalogIn[VAR_ProgressiveId].Man;
			VAR_ManValue	:= HMI_Data.AnalogIn[VAR_ProgressiveId].PV_Man;
		END_IF
	ELSIF (Index < (VAR_ProgressiveId + 4 * HMI_Page.PageNum)) THEN
		IF IN_IOType THEN
			HMI_Data.AnalogOut[VAR_ProgressiveId].Visibility	:= FALSE;
		ELSE
			HMI_Data.AnalogIn[VAR_ProgressiveId].Visibility		:= FALSE;
		END_IF
	END_IF

	VAR_OldPage := HMI_Page.PageNum;

	HMI_Data.ManActive	:= VAR_Man OR HMI_Data.ManActive;

	IF (Index > (4 + 4 * HMI_Page.PageNum)) AND IN_Visibility THEN
		HMI_Data.PageUp.Enable := TRUE;
	END_IF

	IF HMI_Page.PageNum <> 0 THEN
		HMI_Data.PageDown.Enable := TRUE;
	END_IF

	OUT_Man			:= VAR_Man;
	OUT_ManValue	:= VAR_ManValue;
	Index			:= Index + 1;
END_FUNCTION_BLOCK

FUNCTION_BLOCK FB_HMI_ITC_End
	IF IN_IODigAnalog THEN
		VAR_ProgressiveId := INT_TO_UINT(FC_ReminderShift(UINT_TO_INT(Index), 4, 0));
		IF Index < (4 + 4 * HMI_Page.PageNum) THEN
			FOR i := Index TO (4 + Index - VAR_ProgressiveId) DO
				IF IN_IOType THEN
					HMI_Data.AnalogOut[VAR_ProgressiveId + i - Index].Visibility	:= FALSE;
				ELSE
					HMI_Data.AnalogIn[VAR_ProgressiveId + i - Index].Visibility		:= FALSE;
				END_IF
			END_FOR
		END_IF
	ELSE
		VAR_ProgressiveId := INT_TO_UINT(FC_ReminderShift(UINT_TO_INT(Index), 16, 0));
		IF Index < (16 + 16 * HMI_Page.PageNum) THEN
			FOR i := Index TO (16 + Index - VAR_ProgressiveId) DO
				IF IN_IOType THEN
					HMI_Data.DigitalOut[VAR_ProgressiveId + i - Index].Visibility	:= FALSE;
				ELSE
					HMI_Data.DigitalIn[VAR_ProgressiveId + i - Index].Visibility	:= FALSE;
				END_IF
			END_FOR
		END_IF
	END_IF
END_FUNCTION_BLOCK

FUNCTION_BLOCK FB_HMI_ITC_Start
	FOR i := 1 TO 16 DO
		HMI_Data.DigitalIn[i].Visibility	:= FALSE;
		HMI_Data.DigitalOut[i].Visibility	:= FALSE;
		IF i <= 4 THEN
			HMI_Data.AnalogOut[i].Visibility	:= FALSE;
			HMI_Data.AnalogIn[i].Visibility		:= FALSE;
		END_IF
	END_FOR

	HMI_Data.PageDown.Enable	:= FALSE;
	HMI_Data.PageUp.Enable		:= FALSE;
	HMI_Data.ManActive			:= FALSE;

	DigitalIndexIn	:= 1;
	AnalogIndexIn	:= 1;
	DigitalIndexOut	:= 1;
	AnalogIndexOut	:= 1;
END_FUNCTION_BLOCK
```

#### FB_ITCFast.st
```iecst
FUNCTION_BLOCK FB_HMI_ITC_FastDigitalByte
	VAR_ProgressiveId := INT_TO_UINT(FC_ReminderShift(UINT_TO_INT(Index), 16, 0));

	IF IN_ReadOnly OR IN_HMIAutoForce THEN
		VAR_Auto	:= TRUE;
		VAR_Man		:= FALSE;
	END_IF

	IF VAR_OldPage <> HMI_Page.PageNum THEN
		VAR_PageSwitch	:= TRUE;
	END_IF

	IF (Index = (VAR_ProgressiveId + 16 * VAR_OldPage)) AND IN_Visibility THEN
		IF VAR_PageSwitch THEN
			IF IN_IOType THEN
				HMI_Data.DigitalOut[VAR_ProgressiveId].Auto	:= VAR_Auto;
				HMI_Data.DigitalOut[VAR_ProgressiveId].Man	:= VAR_Man;
			ELSE
				HMI_Data.DigitalIn[VAR_ProgressiveId].Auto	:= VAR_Auto;
				HMI_Data.DigitalIn[VAR_ProgressiveId].Man	:= VAR_Man;
			END_IF
			VAR_PageSwitch	:= FALSE;
		END_IF

		IF IN_IOType THEN
			HMI_Data.DigitalOut[VAR_ProgressiveId].Visibility	:= IN_Visibility;
			HMI_Data.DigitalOut[VAR_ProgressiveId].Enable		:= NOT IN_ReadOnly AND NOT IN_HMIAutoForce;
			HMI_Data.DigitalOut[VAR_ProgressiveId].LampState	:= SEL(VAR_Auto, VAR_Man, ITC);
			HMI_Data.DigitalOut[VAR_ProgressiveId].Wait			:= IN_Wait;
			HMI_Data.DigitalOut[VAR_ProgressiveId].Alarm		:= IN_Alarm;
			HMI_Data.DigitalOut[VAR_ProgressiveId].Description	:= IN_Description;

			IF EDGEPOS(HMI_Data.DigitalOut[VAR_ProgressiveId].Auto) THEN
				HMI_Data.DigitalOut[VAR_ProgressiveId].Man := FALSE;
			ELSIF EDGEPOS(HMI_Data.DigitalOut[VAR_ProgressiveId].Man) THEN
				HMI_Data.DigitalOut[VAR_ProgressiveId].Auto := FALSE;
			END_IF

			IF IN_ReadOnly OR IN_HMIAutoForce THEN
				HMI_Data.DigitalOut[VAR_ProgressiveId].Auto	:= TRUE;
				HMI_Data.DigitalOut[VAR_ProgressiveId].Man	:= FALSE;
			END_IF

			VAR_Auto	:= HMI_Data.DigitalOut[VAR_ProgressiveId].Auto;
			VAR_Man		:= HMI_Data.DigitalOut[VAR_ProgressiveId].Man;
		ELSE
			HMI_Data.DigitalIn[VAR_ProgressiveId].Visibility	:= IN_Visibility;
			HMI_Data.DigitalIn[VAR_ProgressiveId].Enable		:= NOT IN_ReadOnly AND NOT IN_HMIAutoForce;
			HMI_Data.DigitalIn[VAR_ProgressiveId].LampState 	:= SEL(VAR_Auto, VAR_Man, ITC);
			HMI_Data.DigitalIn[VAR_ProgressiveId].Wait			:= IN_Wait;
			HMI_Data.DigitalIn[VAR_ProgressiveId].Alarm			:= IN_Alarm;
			HMI_Data.DigitalIn[VAR_ProgressiveId].Description	:= IN_Description;

			IF EDGEPOS(HMI_Data.DigitalIn[VAR_ProgressiveId].Auto) THEN
				HMI_Data.DigitalIn[VAR_ProgressiveId].Man := FALSE;
			ELSIF EDGEPOS(HMI_Data.DigitalIn[VAR_ProgressiveId].Man) THEN
				HMI_Data.DigitalIn[VAR_ProgressiveId].Auto := FALSE;
			END_IF

			IF IN_ReadOnly OR IN_HMIAutoForce THEN
				HMI_Data.DigitalIn[VAR_ProgressiveId].Auto	:= TRUE;
				HMI_Data.DigitalIn[VAR_ProgressiveId].Man	:= FALSE;
			END_IF

			VAR_Auto	:= HMI_Data.DigitalIn[VAR_ProgressiveId].Auto;
			VAR_Man		:= HMI_Data.DigitalIn[VAR_ProgressiveId].Man;
		END_IF
	ELSIF (Index < (VAR_ProgressiveId + 16 * HMI_Page.PageNum)) THEN
		IF IN_IOType THEN
			HMI_Data.DigitalOut[VAR_ProgressiveId].Visibility	:= FALSE;
		ELSE
			HMI_Data.DigitalIn[VAR_ProgressiveId].Visibility	:= FALSE;
		END_IF
	END_IF

	VAR_OldPage := HMI_Page.PageNum;

	HMI_Data.ManActive	:= NOT VAR_Auto OR HMI_Data.ManActive;

	IF (Index > (16 + 16 * HMI_Page.PageNum)) AND IN_Visibility THEN
		HMI_Data.PageUp.Enable := TRUE;
	END_IF

	IF HMI_Page.PageNum <> 0 THEN
		HMI_Data.PageDown.Enable := TRUE;
	END_IF

	OUT_Man			:= NOT VAR_Auto;
	OUT_ManValue	:= VAR_Man;
	Index	:= Index + 1;
END_FUNCTION_BLOCK

FUNCTION_BLOCK FB_HMI_ITC_FastAnalogInt
	VAR_ProgressiveId := INT_TO_UINT(FC_ReminderShift(UINT_TO_INT(Index), 4, 0));

	IF IN_ReadOnly OR IN_HMIAutoForce THEN
		VAR_Man		:= FALSE;
	END_IF

	IF VAR_OldPage <> HMI_Page.PageNum THEN
		VAR_PageSwitch	:= TRUE;
	END_IF

	IF (Index = (VAR_ProgressiveId + 4 * VAR_OldPage)) AND IN_Visibility THEN
		IF VAR_PageSwitch THEN
			IF IN_IOType THEN
				HMI_Data.AnalogOut[VAR_ProgressiveId].Man		:= VAR_Man;
				HMI_Data.AnalogOut[VAR_ProgressiveId].PV_Man	:= INT_TO_REAL(VAR_ManValue);
			ELSE
				HMI_Data.AnalogIn[VAR_ProgressiveId].Man	:= VAR_Man;
				HMI_Data.AnalogIn[VAR_ProgressiveId].PV_Man	:= INT_TO_REAL(VAR_ManValue);
			END_IF
			VAR_PageSwitch	:= FALSE;
		END_IF

		IF IN_IOType THEN
			HMI_Data.AnalogOut[VAR_ProgressiveId].Visibility	:= IN_Visibility;
			HMI_Data.AnalogOut[VAR_ProgressiveId].Enable		:= NOT IN_ReadOnly AND NOT IN_HMIAutoForce;
			HMI_Data.AnalogOut[VAR_ProgressiveId].PV			:= SEL(VAR_Man, INT_TO_REAL(ITC), INT_TO_REAL(VAR_ManValue));
			HMI_Data.AnalogOut[VAR_ProgressiveId].Wait			:= IN_Wait;
			HMI_Data.AnalogOut[VAR_ProgressiveId].Description	:= IN_Description;
			HMI_Data.AnalogOut[VAR_ProgressiveId].Unit			:= IN_Unit;
			HMI_Data.AnalogOut[VAR_ProgressiveId].MaxValue		:= IN_MaxValue;
			HMI_Data.AnalogOut[VAR_ProgressiveId].MinValue		:= IN_MinValue;

			VAR_Man			:= HMI_Data.AnalogOut[VAR_ProgressiveId].Man;
			VAR_ManValue	:= REAL_TO_INT(HMI_Data.AnalogOut[VAR_ProgressiveId].PV_Man);
		ELSE
			HMI_Data.AnalogIn[VAR_ProgressiveId].Visibility		:= IN_Visibility;
			HMI_Data.AnalogIn[VAR_ProgressiveId].Enable			:= NOT IN_ReadOnly AND NOT IN_HMIAutoForce;
			HMI_Data.AnalogIn[VAR_ProgressiveId].PV				:= SEL(VAR_Man, INT_TO_REAL(ITC), INT_TO_REAL(VAR_ManValue));
			HMI_Data.AnalogIn[VAR_ProgressiveId].Wait			:= IN_Wait;
			HMI_Data.AnalogIn[VAR_ProgressiveId].Description	:= IN_Description;
			HMI_Data.AnalogIn[VAR_ProgressiveId].Unit			:= IN_Unit;
			HMI_Data.AnalogIn[VAR_ProgressiveId].MaxValue		:= IN_MaxValue;
			HMI_Data.AnalogIn[VAR_ProgressiveId].MinValue		:= IN_MinValue;

			VAR_Man			:= HMI_Data.AnalogIn[VAR_ProgressiveId].Man;
			VAR_ManValue	:= REAL_TO_INT(HMI_Data.AnalogIn[VAR_ProgressiveId].PV_Man);
		END_IF
	ELSIF (Index < (VAR_ProgressiveId + 4 * HMI_Page.PageNum)) THEN
		IF IN_IOType THEN
			HMI_Data.AnalogOut[VAR_ProgressiveId].Visibility	:= FALSE;
		ELSE
			HMI_Data.AnalogIn[VAR_ProgressiveId].Visibility	:= FALSE;
		END_IF
	END_IF

	VAR_OldPage := HMI_Page.PageNum;

	HMI_Data.ManActive	:= VAR_Man OR HMI_Data.ManActive;

	IF (Index > (4 + 4 * HMI_Page.PageNum)) AND IN_Visibility THEN
		HMI_Data.PageUp.Enable := TRUE;
	END_IF

	IF HMI_Page.PageNum <> 0 THEN
		HMI_Data.PageDown.Enable := TRUE;
	END_IF

	OUT_Man			:= VAR_Man;
	OUT_ManValue	:= VAR_ManValue;
	Index	:= Index + 1;
END_FUNCTION_BLOCK

FUNCTION_BLOCK FB_HMI_ITC_FastAnalogDInt
	VAR_ProgressiveId := INT_TO_UINT(FC_ReminderShift(UINT_TO_INT(Index), 4, 0));

	IF IN_ReadOnly OR IN_HMIAutoForce THEN
		VAR_Man		:= FALSE;
	END_IF

	IF VAR_OldPage <> HMI_Page.PageNum THEN
		VAR_PageSwitch	:= TRUE;
	END_IF

	IF (Index = (VAR_ProgressiveId + 4 * VAR_OldPage)) AND IN_Visibility THEN
		IF VAR_PageSwitch THEN
			IF IN_IOType THEN
				HMI_Data.AnalogOut[VAR_ProgressiveId].Man		:= VAR_Man;
				HMI_Data.AnalogOut[VAR_ProgressiveId].PV_Man	:= DINT_TO_REAL(VAR_ManValue);
			ELSE
				HMI_Data.AnalogIn[VAR_ProgressiveId].Man	:= VAR_Man;
				HMI_Data.AnalogIn[VAR_ProgressiveId].PV_Man	:= DINT_TO_REAL(VAR_ManValue);
			END_IF
			VAR_PageSwitch	:= FALSE;
		END_IF

		IF IN_IOType THEN
			HMI_Data.AnalogOut[VAR_ProgressiveId].Visibility	:= IN_Visibility;
			HMI_Data.AnalogOut[VAR_ProgressiveId].Enable		:= NOT IN_ReadOnly AND NOT IN_HMIAutoForce;
			HMI_Data.AnalogOut[VAR_ProgressiveId].PV			:= SEL(VAR_Man, DINT_TO_REAL(ITC), DINT_TO_REAL(VAR_ManValue));
			HMI_Data.AnalogOut[VAR_ProgressiveId].Wait			:= IN_Wait;
			HMI_Data.AnalogOut[VAR_ProgressiveId].Description	:= IN_Description;
			HMI_Data.AnalogOut[VAR_ProgressiveId].Unit			:= IN_Unit;
			HMI_Data.AnalogOut[VAR_ProgressiveId].MaxValue		:= IN_MaxValue;
			HMI_Data.AnalogOut[VAR_ProgressiveId].MinValue		:= IN_MinValue;

			VAR_Man			:= HMI_Data.AnalogOut[VAR_ProgressiveId].Man;
			VAR_ManValue	:= REAL_TO_INT(HMI_Data.AnalogOut[VAR_ProgressiveId].PV_Man);
		ELSE
			HMI_Data.AnalogIn[VAR_ProgressiveId].Visibility		:= IN_Visibility;
			HMI_Data.AnalogIn[VAR_ProgressiveId].Enable			:= NOT IN_ReadOnly AND NOT IN_HMIAutoForce;
			HMI_Data.AnalogIn[VAR_ProgressiveId].PV				:= SEL(VAR_Man, DINT_TO_REAL(ITC), DINT_TO_REAL(VAR_ManValue));
			HMI_Data.AnalogIn[VAR_ProgressiveId].Wait			:= IN_Wait;
			HMI_Data.AnalogIn[VAR_ProgressiveId].Description	:= IN_Description;
			HMI_Data.AnalogIn[VAR_ProgressiveId].Unit			:= IN_Unit;
			HMI_Data.AnalogIn[VAR_ProgressiveId].MaxValue		:= IN_MaxValue;
			HMI_Data.AnalogIn[VAR_ProgressiveId].MinValue		:= IN_MinValue;

			VAR_Man			:= HMI_Data.AnalogIn[VAR_ProgressiveId].Man;
			VAR_ManValue	:= REAL_TO_INT(HMI_Data.AnalogIn[VAR_ProgressiveId].PV_Man);
		END_IF
	ELSIF (Index < (VAR_ProgressiveId + 4 * HMI_Page.PageNum)) THEN
		IF IN_IOType THEN
			HMI_Data.AnalogOut[VAR_ProgressiveId].Visibility	:= FALSE;
		ELSE
			HMI_Data.AnalogIn[VAR_ProgressiveId].Visibility	:= FALSE;
		END_IF
	END_IF

	VAR_OldPage := HMI_Page.PageNum;

	HMI_Data.ManActive	:= VAR_Man OR HMI_Data.ManActive;

	IF (Index > (4 + 4 * HMI_Page.PageNum)) AND IN_Visibility THEN
		HMI_Data.PageUp.Enable := TRUE;
	END_IF

	IF HMI_Page.PageNum <> 0 THEN
		HMI_Data.PageDown.Enable := TRUE;
	END_IF

	OUT_Man			:= VAR_Man;
	OUT_ManValue	:= VAR_ManValue;
	Index	:= Index + 1;
END_FUNCTION_BLOCK
```

#### FB_Counter.st
```iecst
FUNCTION_BLOCK FB_Counter
	IF(IN_Clock1Hz) AND IN_TimeCondition THEN
		IN_OUT_CounterPartialStruct.CounterTime.Sec	:= IN_OUT_CounterPartialStruct.CounterTime.Sec + 1;
		IF (IN_OUT_CounterPartialStruct.CounterTime.Sec >= 60) THEN
			IN_OUT_CounterPartialStruct.CounterTime.Sec	:= 0;
			IN_OUT_CounterPartialStruct.CounterTime.Min	:= IN_OUT_CounterPartialStruct.CounterTime.Min + 1;
			IF IN_OUT_CounterPartialStruct.CounterTime.Min >= 60 THEN
				IN_OUT_CounterPartialStruct.CounterTime.Min	:= 0;
				IN_OUT_CounterPartialStruct.CounterTime.Hour	:= IN_OUT_CounterPartialStruct.CounterTime.Hour + 1;
				IF IN_OUT_CounterPartialStruct.CounterTime.Hour >= 24 THEN
					IN_OUT_CounterPartialStruct.CounterTime.Hour	:= 0;
					IN_OUT_CounterPartialStruct.CounterTime.Day	:= IN_OUT_CounterPartialStruct.CounterTime.Day + 1;
				END_IF
			END_IF
		END_IF

		IN_OUT_CounterTotalStruct.CounterTime.Sec	:= IN_OUT_CounterTotalStruct.CounterTime.Sec + 1;
		IF (IN_OUT_CounterTotalStruct.CounterTime.Sec >= 60) THEN
			IN_OUT_CounterTotalStruct.CounterTime.Sec	:= 0;
			IN_OUT_CounterTotalStruct.CounterTime.Min	:= IN_OUT_CounterTotalStruct.CounterTime.Min + 1;
			IF IN_OUT_CounterTotalStruct.CounterTime.Min >= 60 THEN
				IN_OUT_CounterTotalStruct.CounterTime.Min	:= 0;
				IN_OUT_CounterTotalStruct.CounterTime.Hour	:= IN_OUT_CounterTotalStruct.CounterTime.Hour + 1;
				IF IN_OUT_CounterTotalStruct.CounterTime.Hour >= 24 THEN
					IN_OUT_CounterTotalStruct.CounterTime.Hour	:= 0;
					IN_OUT_CounterTotalStruct.CounterTime.Day	:= IN_OUT_CounterTotalStruct.CounterTime.Day + 1;
				END_IF
			END_IF
		END_IF
	END_IF

	IF IN_IncrementCondition THEN
		tempReal := tempReal + IN_PulseWeight;
		IF tempReal >= 1.0 THEN
			IN_OUT_CounterPartialStruct.CounterValue	:= IN_OUT_CounterPartialStruct.CounterValue + TRUNC(tempReal);
			IN_OUT_CounterTotalStruct.CounterValue		:= IN_OUT_CounterTotalStruct.CounterValue 	+ TRUNC(tempReal);
			tempReal := tempReal - (TRUNC(tempReal));
		END_IF
	END_IF

	IF IN_Reset THEN
		IN_OUT_CounterPartialStruct.CounterTime.Sec		:= 0;
		IN_OUT_CounterPartialStruct.CounterTime.Min		:= 0;
		IN_OUT_CounterPartialStruct.CounterTime.Hour	:= 0;
		IN_OUT_CounterPartialStruct.CounterTime.Day		:= 0;
		IN_OUT_CounterPartialStruct.CounterValue		:= 0;
		IN_OUT_CounterPartialStruct.StartDate			:= DT_TO_DINT(IN_Date);
	ELSIF IN_OUT_CounterPartialStruct.StartDate = 0 THEN
		IN_OUT_CounterPartialStruct.StartDate		:= DT_TO_DINT(IN_Date);
	ELSIF IN_OUT_CounterTotalStruct.StartDate	= 0 THEN
		IN_OUT_CounterTotalStruct.StartDate		:= DT_TO_DINT(IN_Date);
	END_IF
END_FUNCTION_BLOCK
```

#### FC_Counter.st
```iecst
FUNCTION FC_Counter
	IF(IN_Clock1Hz) AND IN_TimeCondition THEN
		FC_Counter	:= TRUE;
		IN_OUT_CounterPartialStruct.CounterTime.Sec	:= IN_OUT_CounterPartialStruct.CounterTime.Sec + 1;
		IF (IN_OUT_CounterPartialStruct.CounterTime.Sec >= 60) THEN
			IN_OUT_CounterPartialStruct.CounterTime.Sec	:= 0;
			IN_OUT_CounterPartialStruct.CounterTime.Min	:= IN_OUT_CounterPartialStruct.CounterTime.Min + 1;
			IF IN_OUT_CounterPartialStruct.CounterTime.Min >= 60 THEN
				IN_OUT_CounterPartialStruct.CounterTime.Min	:= 0;
				IN_OUT_CounterPartialStruct.CounterTime.Hour	:= IN_OUT_CounterPartialStruct.CounterTime.Hour + 1;
				IF IN_OUT_CounterPartialStruct.CounterTime.Hour >= 24 THEN
					IN_OUT_CounterPartialStruct.CounterTime.Hour	:= 0;
					IN_OUT_CounterPartialStruct.CounterTime.Day	:= IN_OUT_CounterPartialStruct.CounterTime.Day + 1;
				END_IF
			END_IF
		END_IF

		IN_OUT_CounterTotalStruct.CounterTime.Sec	:= IN_OUT_CounterTotalStruct.CounterTime.Sec + 1;
		IF (IN_OUT_CounterTotalStruct.CounterTime.Sec >= 60) THEN
			IN_OUT_CounterTotalStruct.CounterTime.Sec	:= 0;
			IN_OUT_CounterTotalStruct.CounterTime.Min	:= IN_OUT_CounterTotalStruct.CounterTime.Min + 1;
			IF IN_OUT_CounterTotalStruct.CounterTime.Min >= 60 THEN
				IN_OUT_CounterTotalStruct.CounterTime.Min	:= 0;
				IN_OUT_CounterTotalStruct.CounterTime.Hour	:= IN_OUT_CounterTotalStruct.CounterTime.Hour + 1;
				IF IN_OUT_CounterTotalStruct.CounterTime.Hour >= 24 THEN
					IN_OUT_CounterTotalStruct.CounterTime.Hour	:= 0;
					IN_OUT_CounterTotalStruct.CounterTime.Day	:= IN_OUT_CounterTotalStruct.CounterTime.Day + 1;
				END_IF
			END_IF
		END_IF
	END_IF

	IF IN_IncrementCondition THEN
		FC_Counter	:= TRUE;
		IN_OUT_CounterPartialStruct.CounterValue	:= IN_OUT_CounterPartialStruct.CounterValue + 1;
		IN_OUT_CounterTotalStruct.CounterValue		:= IN_OUT_CounterTotalStruct.CounterValue + 1;
	END_IF

	IF IN_Reset THEN
		FC_Counter	:= TRUE;
		IN_OUT_CounterPartialStruct.CounterTime.Sec		:= 0;
		IN_OUT_CounterPartialStruct.CounterTime.Min		:= 0;
		IN_OUT_CounterPartialStruct.CounterTime.Hour	:= 0;
		IN_OUT_CounterPartialStruct.CounterTime.Day		:= 0;
		IN_OUT_CounterPartialStruct.CounterValue		:= 0;
		IN_OUT_CounterPartialStruct.StartDate			:= DT_TO_DINT(IN_Date);
	ELSIF IN_OUT_CounterPartialStruct.StartDate = 0 THEN
		IN_OUT_CounterPartialStruct.StartDate		:= DT_TO_DINT(IN_Date);
	ELSIF IN_OUT_CounterTotalStruct.StartDate	= 0 THEN
		IN_OUT_CounterTotalStruct.StartDate		:= DT_TO_DINT(IN_Date);
	END_IF
END_FUNCTION
```

#### FC_Timer.st
```iecst
FUNCTION FC_IncTimer
	IF IN_Reset THEN
		FC_IncTimer	:= TRUE;
		IN_OUT_CounterStruct.Sec	:= 0;
		IN_OUT_CounterStruct.Min	:= 0;
		IN_OUT_CounterStruct.Hour	:= 0;
		IN_OUT_CounterStruct.Day	:= 0;
	ELSIF(IN_Clock1Hz) AND IN_Condition THEN
		FC_IncTimer	:=	TRUE;
		IN_OUT_CounterStruct.Sec	:= IN_OUT_CounterStruct.Sec + 1;
		IF (IN_OUT_CounterStruct.Sec >= 60) THEN
			IN_OUT_CounterStruct.Sec	:= 0;
			IN_OUT_CounterStruct.Min	:= IN_OUT_CounterStruct.Min + 1;
			IF IN_OUT_CounterStruct.Min >= 60 THEN
				IN_OUT_CounterStruct.Min	:= 0;
				IN_OUT_CounterStruct.Hour	:= IN_OUT_CounterStruct.Hour + 1;
				IF IN_OUT_CounterStruct.Hour >= 24 THEN
					IN_OUT_CounterStruct.Hour	:= 0;
					IN_OUT_CounterStruct.Day	:= IN_OUT_CounterStruct.Day + 1;
				END_IF
			END_IF
		END_IF
	ELSE
		FC_IncTimer	:= FALSE;
	END_IF
END_FUNCTION

FUNCTION FC_MacaoTimer
	IF IN_Reset THEN
		IN_OUT_Counter	:= 0;
	ELSIF IN_Clock1Hz AND IN_Condition THEN
		IN_OUT_Counter	:= IN_OUT_Counter + 1;
	END_IF
	FC_MacaoTimer := TRUE;
END_FUNCTION
```

#### FC_Parity.st
```iecst
FUNCTION FC_Parity
	FC_Parity := NOT IN_Value.0;
END_FUNCTION
```

#### FC_Reminder.st
```iecst
(* Reminder With Minimum Value *)
FUNCTION FC_ReminderShift
	LocalDivisor	:= SEL(Divisor<>0, 1, Divisor);

	ReminderA	:= (Dividend - ((Dividend / LocalDivisor) * LocalDivisor));
	ReminderB	:= (ReminderA + Divisor - ((ReminderA + LocalDivisor) / LocalDivisor) * LocalDivisor);
	ReminderC	:= (ReminderB + Start - ((ReminderB + Start) / LocalDivisor) * LocalDivisor);

	FC_ReminderShift	:= SEL(ReminderC <> 0, LocalDivisor, ReminderC);
END_FUNCTION
```

#### FC_SpeedCheck.st
```iecst
FUNCTION FC_SpeedCheck
	CASE IN_Mode OF
		CST_EQ:	(* Actual speed equal to requested *)
			FC_SpeedCheck := (IN_SpeedAct >= (IN_SpeedReq * 0.9)) AND (IN_SpeedAct <= (IN_SpeedReq / 0.9));

		CST_GE:	(* Actual speed greater then requested *)
			FC_SpeedCheck := IN_SpeedAct >= IN_SpeedReq * 0.9;

		CST_LE:	(* Actual speed lower then requested *)
			FC_SpeedCheck := IN_SpeedAct <= IN_SpeedReq / 0.9;

		CST_GT:	(* Actual speed greater then requested *)
			FC_SpeedCheck := IN_SpeedAct > IN_SpeedReq * 0.9;

		CST_LT:	(* Actual speed lower then requested *)
			FC_SpeedCheck := IN_SpeedAct < IN_SpeedReq / 0.9;

		ELSE
			FC_SpeedCheck := FALSE;
	END_CASE
END_FUNCTION
```

#### LevelVariation.st
```iecst
(********************************************************************
 * COPYRIGHT -- Sidel S.p.A.
 ********************************************************************
 * Program: PC
 * File: Balayage_Flow_Contr.st
 * Author: Marco.Nicoli
 * Created: December 10, 2012
 ********************************************************************
 * Implementation of program PC
 ********************************************************************)

(*  *)
FUNCTION_BLOCK LevelVariation
	VAR_RTInfo(enable:=TRUE);
	VAR_Cycle:=	UDINT_TO_REAL(VAR_RTInfo.cycle_time)/1000000; //TASK CYCLE TIME EXPRESS IN µsec . VAR_Cycle IS CONVERTED IN s

	IF IN_Enable THEN
		IF Timer > IN_ControlTime THEN
			DeltaVolume := (IN_TankVolumePV - OldVolume);						//LEVEL VARIATION CONTROL
			IF DeltaVolume < -1.0 THEN
				AbsoluteError := AbsoluteError + ABS (DeltaVolume);				//WHEN VARIATION IS NEGATIVE THE ERROR INCREASE
				RestoreTime	  := 0.0;											//WHEN VARIATION IS NEGATIVE RESTORE TIME IS RESET
				RestoreError  := 0.0;											//WHEN VARIATION IS NEGATIVE RESTORE ERROR IS RESET
			ELSIF OUT_High THEN
				RestoreTime	:= LIMIT (0.0,RestoreTime + 1.0,RestoreTimeLimit);	//WHEN VARIATION IS POSITIVE RESTORE TIME INCREASE
				RestoreError:= 0.0;												//WHEN VARIATION IS NEGATIVE RESTORE ERROR IS RESET
			ELSE
				RestoreError := LIMIT (0.0,RestoreError + 1.0,RestoreErrorLimit); //WHEN NO ACTION BEFORE INCREASE ERROR
			END_IF

			IF RestoreTime >= RestoreTimeLimit THEN								//WHEN RESTORE TIME LIMIT REACHED VARIATION IS STEADY
				AbsoluteError	:= 0.0;											//RestoreTimeLimit = 50.0 -> Timer x 50 -> 200ms x 50 = 10s
				RestoreTime 	:= 0.0;
			END_IF

			IF RestoreError >= RestoreErrorLimit THEN 							//WHEN RESTORE ERROR IS REACHED ERROR IS RESET
				AbsoluteError   := 0.0;               							//RestoreErrorLimit = 50.0 -> Timer x 50 -> 200ms x 50 = 10s
				RestoreError    := 0.0;
			END_IF

			OldVolume	:= IN_TankVolumePV;										//ACTUAL VOLUME UPDATE
			Timer		:= 0.0;													//CYCLE TIME RESTART
		ELSE
			Timer := Timer + VAR_Cycle ;										//CYCLE TIME UPDATE
		END_IF
	ELSE
		Timer 			:= 0.0;
		AbsoluteError 	:= 0.0;
		RestoreTime 	:= 0.0;
		RestoreError    := 0.0;
		OldVolume 		:= IN_TankVolumePV;
	END_IF

	OUT_High	:= AbsoluteError > 3.0;											//HIGH FLOW REQUEST DUE TO PERSISTENT NEGATIVE VARIATION
	OUT_Low 	:= NOT OUT_High;												//LOW FLOW REQUEST DUE TO VARIATION IN TOLERANCE

END_FUNCTION_BLOCK
```

#### LftConAirPress.st
```iecst
FUNCTION LftConAirPressSp
	VAR_PistonSurface 	:= amPI * (EXPT(CST_PistonDiameterExt, 2) - EXPT(CST_PistonDiameterInt, 2)) / 4.0;
	VAR_DeltaPProduct 	:= (EXPT(57.0, 2) - EXPT(RcpCanDiameter, 2)) * amPI / 4.0 * RcpPressureSp / 10.0;
	VAR_DeltaPrexPist  	:= (ABS(VAR_DeltaPProduct * 1000000.0 / VAR_PistonSurface / 100000.0)) * BOOL_TO_REAL((RcpCanDiameter > 57.0));
	VAR_PbasePiston 	:= CST_PistonSpringStrengthRse / (VAR_PistonSurface / 100.0) / 10;
	LftConAirPressSp	:= VAR_PbasePiston + VAR_DeltaPrexPist + 1.5;
END_FUNCTION
```

#### RCP_Management.st
```iecst
FUNCTION_BLOCK RCP_Management
	IF NOT VAR_FirstCycle THEN
		IF (memcmp(IN_AdrPLCRecipe, IN_AdrHMIRecipe, IN_SizePLCRecipe) <> 0) OR (memcmp(IN_AdrHMIRecipe, IN_AdrPLCRecipe, IN_SizeHMIRecipe) <> 0) THEN
			OUT_ParameterError := TRUE;
			RETURN;
		ELSE
			VAR_FirstCycle := TRUE;
		END_IF
	END_IF

	TMR_tonRCP_WaitStart.IN			:= FALSE;
	TMR_tonRCP_DownloadTimeOut.IN	:= FALSE;

	CASE OUT_Step OF

		Wait_Download:
			RCP_Manag.RequestedRecipeName	:= IN_RequestedRCP;
			TMR_tonRCP_WaitStart.IN			:= IN_DownloadRequest OR RCP_Manag.Started;
			TMR_tonRCP_WaitStart.PT			:= t#500ms;

			IF TMR_tonRCP_WaitStart.Q THEN
				OUT_Step := Download_Request;
			END_IF

			IF RCP_Manag.EditOnlineActive THEN
				OUT_Step := Edit_Online;
			END_IF

		Download_Request:
			RCP_Manag.RequestedRecipeName 	:= IN_RequestedRCP;
			RCP_Manag.DownloadRequest		:= IN_DownloadRequest;

			IF (RCP_Manag.Started AND RCP_Manag.Ended) THEN
				OUT_Step := Copy_To_Internal;
			END_IF

			TMR_tonRCP_DownloadTimeOut.IN	:= NOT RCP_Manag.Ended OR (NOT RCP_Manag.Started AND RCP_Manag.Ended);
			TMR_tonRCP_DownloadTimeOut.PT	:= t#10s;

			IF TMR_tonRCP_DownloadTimeOut.Q THEN
				OUT_Step := Download_Error;
			END_IF

		Copy_To_Internal:
			RCP_Manag.DownloadRequest := FALSE;

			IF (memcmp(IN_AdrPLCRecipe,IN_AdrHMIRecipe,IN_SizePLCRecipe) <> 0) THEN
				memcpy(IN_AdrPLCRecipe,IN_AdrHMIRecipe,IN_SizePLCRecipe);
			END_IF

			IF IN_DownloadRequest THEN
				IF (IN_RequestedRCP = RCP_Manag.ActiveRecipeName) THEN	// Check Request Recipe Name
					IF (memcmp(IN_AdrPLCRecipe,IN_AdrHMIRecipe,IN_SizePLCRecipe) = 0) THEN
						OUT_Step := Download_Done;
					END_IF
				END_IF
			ELSE
				OUT_Step := Download_Done;
			END_IF

			TMR_tonRCP_DownloadTimeOut.IN := (IN_RequestedRCP <> RCP_Manag.ActiveRecipeName);
			TMR_tonRCP_DownloadTimeOut.PT := t#5s;

			IF TMR_tonRCP_DownloadTimeOut.Q THEN
				OUT_Step := Download_Error;
			END_IF

		Download_Done:
			RCP_Manag.Received	:= TRUE;
			OUT_RecipeLoaded	:= TRUE;

			IF (NOT RCP_Manag.Ended AND NOT (IN_DownloadRequest OR RCP_Manag.Started)) THEN
				OUT_Step := Clear_Cmd;
			END_IF

		Clear_Cmd:
			RCP_Manag.Received := FALSE;
			RCP_Manag.RequestedRecipeName := '';
			OUT_Step := Wait_Download;

		Edit_Online:
			IF RCP_Manag.EditOnlineActive THEN
				IF (memcmp(IN_AdrPLCRecipe,IN_AdrHMIRecipe,IN_SizePLCRecipe) <> 0) THEN
					memcpy(IN_AdrPLCRecipe,IN_AdrHMIRecipe,IN_SizePLCRecipe);
				END_IF
			ELSE
				OUT_Step := Clear_Cmd;
			END_IF

		Download_Error:
			RCP_Manag.Received := FALSE;
			RCP_Manag.DownloadRequest := FALSE;
			RCP_Manag.Started := FALSE;
			RCP_Manag.Ended := FALSE;
			RCP_Manag.RequestedRecipeName := '';

			TMR_tonRCP_WaitRestart.IN := IN_DownloadRequest OR RCP_Manag.Started;
			TMR_tonRCP_WaitRestart.PT := t#3s;

			IF TMR_tonRCP_WaitRestart.Q THEN
				OUT_Step := Download_Request;
			END_IF

			IF NOT IN_DownloadRequest AND NOT RCP_Manag.Started THEN
				OUT_Step := Wait_Download;
			END_IF
	END_CASE

	IF OUT_Step <> VAR_Step_old THEN
		TMR_tonRCP_WaitStart.IN			:= FALSE;
		TMR_tonRCP_DownloadTimeOut.IN	:= FALSE;
		VAR_Step_old := OUT_Step;
	END_IF

	TMR_tonRCP_WaitStart();
	TMR_tonRCP_DownloadTimeOut();
	TMR_tonRCP_WaitRestart();//v1.7.6
END_FUNCTION_BLOCK
```

#### PID_FB.st - PID calculation
```iecst
FUNCTION_BLOCK PID_Cont
	VAR_RTInfo(enable:=TRUE);
	VAR_CycleCounter	:= MAX(1, VAR_CycleCounter + 1);

	TON_Cycle(	IN := TRUE,
				PT := IN_CycleTime - UDINT_TO_TIME(VAR_RTInfo.cycle_time / 1000));

	IF NOT TON_Cycle.Q THEN
		RETURN;
	END_IF

	VAR_CycleTime	:= (UDINT_TO_REAL(VAR_RTInfo.cycle_time) * VAR_CycleCounter) / 1000000.0;
	VAR_CycleCounter 	:= 0.0;
	memset(ADR(TON_Cycle), 0, SIZEOF(TON_Cycle));

	(*****************************************************************)
	(*************************SP MANAGE*******************************)
	(*****************************************************************)
	IF NOT VAR_FirstCycle THEN
		VAR_FirstCycle	:= TRUE;
		HMI.SPLocal		:= FALSE;
		OUT		:= 0.0;
		OUT_P	:= 0.0;
		OUT_I	:= 0.0;
		OUT_D	:= 0.0;
	END_IF

	IF EDGE(HMI.SPLocal) OR EDGEPOS(IN_Auto) THEN
		VAR_SlewInit	:= TRUE;
	END_IF

	IF VAR_SlewInit AND HMI.SPLocal THEN
		HMI.PV		:= IN_PV;
		LCRRamp.x	:= MIN(IN_PV, HMI.SP_Local);
		LCRRamp.set	:= TRUE;
	ELSIF VAR_SlewInit AND IN_Auto THEN
		HMI.PV		:= IN_PV;
		LCRRamp.x	:= MIN(IN_PV, IN_AutoSP);
		LCRRamp.set	:= TRUE;
	ELSIF HMI.SPLocal THEN
		HMI.PV		:= IN_PV;
		LCRRamp.x	:= HMI.SP_Local;
		LCRRamp.set	:= NOT HMI.ConfigSlewPresent;
	ELSIF IN_Auto THEN
		HMI.PV		:= IN_PV;
		LCRRamp.x	:= IN_AutoSP;
		LCRRamp.set := NOT HMI.ConfigSlewPresent;
	ELSE
		HMI.PV		:= 0.0;
		LCRRamp.x	:= 0.0;
		LCRRamp.set	:= TRUE;
	END_IF

	IF VAR_SlewInit AND LCRRamp.x_reached THEN
		VAR_SlewInit := FALSE;
	END_IF

	LCRRamp(
		enable	:= TRUE,
		dy_up	:= MAX(0.01, IN_SPSlew),
		dy_down := MAX(0.01, IN_SPSlew),
		y_min	:= 0.0,
		y_max	:= IN_MaxScale,
		y_set	:= LCRRamp.x
		);

	VAR_SPRamped := LCRRamp.y;

	(*****************************************************************)
	(***********************PID CONTROL*******************************)
	(*****************************************************************)
	IF IN_ConfigEngValue THEN
		LCRLimScal_PV(
			x	:= IN_PV,
			x1	:= 0.0,
			y1	:= 0.0,
			x2	:= IN_MaxScale,
			y2	:= 100.0
			);
		VAR_PV	:= LCRLimScal_PV.y;

		LCRLimScal_SP(
			x	:= VAR_SPRamped,
			x1	:= 0.0,
			y1	:= 0.0,
			x2	:= IN_MaxScale,
			y2	:= 100.0
			);
		VAR_SP	:= LCRLimScal_SP.y;
	ELSE
		VAR_SP	:= VAR_SPRamped;
		VAR_PV	:= IN_PV;
	END_IF

	IF IN_Reverse THEN
		OUT_Error := (VAR_PV - VAR_SP);
	ELSE
		OUT_Error := (VAR_SP - VAR_PV);
	END_IF

	(*****************************************************************)
	(********************PROPORTIONAL FACTOR**************************)
	(*****************************************************************)
	IF IN_Gain = 0 THEN
		VAR_GainError := OUT_Error;
	ELSE
		VAR_GainError := OUT_Error * IN_Gain;
	END_IF

	IF (IN_Auto OR HMI.SPLocal) THEN
		VAR_Proportional := VAR_GainError;
	ELSE
		VAR_Proportional := 0.0;
	END_IF

	OUT_P := VAR_Proportional;

	(*****************************************************************)
	(***********************INTEGRAL FACTOR***************************)
	(*****************************************************************)
	VAR_IntegralSaturation := (((OUT_P + OUT_I + OUT_D + IN_Disv) > IN_OutMax) AND OUT_Error > 0) OR (((OUT_P + OUT_I + OUT_D + IN_Disv) < IN_OutMin) AND OUT_Error < 0);
	VAR_IntegralBlock := IN_IntHold OR NOT (IN_Auto OR HMI.SPLocal) OR VAR_IntegralSaturation;  // integral block if saturated (anti wind up)

	VAR_Integral.IN_IntCycle := VAR_CycleTime;

	IF (IN_Auto OR HMI.SPLocal) AND IN_TI > 0 AND NOT IN_TIInit THEN
		IF EDGEPOS(IN_Auto OR HMI.SPLocal)THEN
			IF OUT > 0 THEN
				VAR_IntegralOut := OUT - OUT_P - IN_Disv;    (* Bumpless - Inizilize the Integral Component when the PID is setted in auto again *)
				VAR_Integral.IN_NewValue := VAR_IntegralOut;
				VAR_Integral(OUT_Integral := VAR_IntegralOut);
			END_IF
		ELSIF NOT VAR_IntegralBlock THEN
			VAR_Integral.IN_NewValue := VAR_GainError / IN_TI;
			//	VAR_IntegralOut := VAR_IntegralOut;
			IF VAR_Integral.IN_IntCycle > 0 THEN
				VAR_Integral(OUT_Integral := VAR_IntegralOut);
			END_IF
		END_IF
	ELSE
		IF IN_TIInit THEN
			VAR_IntegralOut := IN_TIInitValue;
		ELSE
			VAR_IntegralOut := 0.0;
		END_IF
	END_IF

	OUT_I := LIMIT((IN_OutMax * -1.0), VAR_IntegralOut, IN_OutMax);

	(*****************************************************************)
	(**********************DERIVATIVE FACTOR**************************)
	(*****************************************************************)
	IF (IN_Auto OR HMI.SPLocal) AND IN_TD >0 AND VAR_CycleTime > 0 THEN
		VAR_Derivative := ( VAR_GainError - VAR_OldError ) * IN_TD / VAR_CycleTime;
	ELSE
		VAR_Derivative := 0.0;
	END_IF
	VAR_OldError := VAR_GainError;

	OUT_D := VAR_Derivative;

	(*****************************************************************)
	(************************OUT CALCOLATION**************************)
	(*****************************************************************)
	IF HMI.Enable AND IN_ConfigPresent THEN
		OUT:= LIMIT(IN_OutMin, OUT_P + OUT_I + OUT_D + IN_Disv, IN_OutMax);
	ELSIF IN_FixOut THEN
		OUT:= LIMIT(IN_OutMin, IN_FixOutValue, IN_OutMax);
	ELSE
		OUT:= 0.0;
	END_IF

	(*****************************************************************)
	(*******************************HMI*******************************)
	(*****************************************************************)
	HMI.Enable			:= IN_Auto OR HMI.SPLocal;
	HMI.Mode			:= NOT HMI.SPLocal;
	HMI.SP_SlewRunning	:= LCRRamp.enable AND NOT LCRRamp.x_reached;

	HMI.ConfigPresent		:= IN_ConfigPresent;
	HMI.ConfigSlewPresent	:= IN_Slew;

	OUT_ActSP			:= VAR_SPRamped;
	HMI.SP_Actual		:= OUT_ActSP;
	HMI.SP_Target		:= IN_AutoSP;
	HMI.SP_Obtained		:= (IN_PV < (IN_AutoSP + IN_MaxDev)) AND (IN_PV > (IN_AutoSP - IN_MinDev));
	HMI.FF_OUT			:= IN_Disv;
	HMI.OUT				:= OUT;
END_FUNCTION_BLOCK

FUNCTION_BLOCK Integral
	OUT_Integral := OUT_Integral + ( VAR_OldValue + (IN_NewValue -  VAR_OldValue ) * 0.5 ) * IN_IntCycle;
	VAR_OldValue := IN_NewValue;
END_FUNCTION_BLOCK
```

#### Siko_Management.st
```iecst
(********************************************************************
 * COPYRIGHT -- Sidel
 ********************************************************************
 * Library: SIDEL
 * File: Siko_Management.st
 * Author: 100383
 * Created: November 23, 2015
 ********************************************************************
 * Implementation of library SIDEL
 ********************************************************************)

FUNCTION_BLOCK Siko_Management

	IF IN_SikoData.AbortPositioning AND NOT IN_SikoData.PositioningInProgress THEN
		IN_SikoData.AbortPositioning := FALSE;
	END_IF

	IN_SikoData.Enable := IN_HMI_MotEnable;

	IN_SikoData.StartWrite	:= IN_HMI_StartWrite;
	IN_SikoData.Calibrate	:= IN_HMI_Calibrate;
	IN_SikoData.StartRead	:= IN_HMI_StartRead;

	StepTimer();

	CASE IN_Mode OF
		0:
			IN_SikoData.TargetPos	:= IN_SikoData.CurrentPos;

		1:
			IN_SikoData.TargetPos	:= IN_PosProduction;

		2:
			IN_SikoData.TargetPos	:= IN_PosCleaning;

		ELSE
			IN_Mode := 0;
			Status	:= 0;

	END_CASE

	CASE Status OF
		0:		//Ready IDLE
			OUT_Running			:= FALSE;
			OUT_Done			:= FALSE;
			OUT_PositionError	:= FALSE;

			IN_SikoData.StartPositioning := FALSE;

			IN_SikoData.JogBackward    := IN_HMI_JogBackward AND NOT IN_HMI_MoveAt AND IN_HMI_ManualEnable;
			IN_SikoData.JogForward     := IN_HMI_JogForward  AND NOT IN_HMI_MoveAt AND IN_HMI_ManualEnable;

			StepTimer.IN := FALSE;
			StepTimer.PT := t#0s;

			IF IN_Mode = 1  AND NOT IN_HMI_ManualEnable THEN
				Status := 100;
			END_IF

			IF IN_Mode = 2 AND NOT IN_HMI_ManualEnable THEN
				Status := 200;
			END_IF

			IF IN_Mode = 0 AND EDGENEG(IN_HMI_MoveAt) AND NOT IN_HMI_JogForward AND NOT IN_HMI_JogBackward AND IN_HMI_ManualEnable THEN
				IN_SikoData.TargetPos := IN_PosManualSP;
				Status	:= 10;
			END_IF

		10:		//Manual positioning
			OUT_Running			:= FALSE;
			OUT_Done			:= FALSE;
			OUT_PositionError	:= FALSE;

			StepTimer.IN	:= TRUE;
			StepTimer.PT	:= t#240s;

			IN_SikoData.StartPositioning	:=	IN_SikoData.CalibrationDone			AND NOT IN_SikoData.OnError					AND NOT
												IN_SikoData.CommunicationFault		AND NOT IN_SikoData.MotorDisabled			AND IN_SikoData.EmergencyOkFbk	AND NOT
												IN_SikoData.TargetOutsideSwLimit	AND NOT IN_SikoData.DeviceOutsideSwLimit;

			IN_SikoData.TargetPos			:= IN_PosManualSP;

			//Motor in position
			IF IN_SikoData.InPosition THEN
				IN_SikoData.StartPositioning := FALSE;
				StepTimer.IN := FALSE;
				Status := 0;
			END_IF

			//Timeout positioning or change modality
			IF StepTimer.Q OR EDGEPOS(IN_HMI_MoveAt) OR NOT IN_HMI_ManualEnable OR IN_Mode <> 0 THEN
				IN_SikoData.StartPositioning := FALSE;
				IN_SikoData.AbortPositioning := TRUE;
				StepTimer.IN := FALSE;
				Status := 20;
			END_IF

		20:		//Abort command. Wait 0.5s motor stop before changing mode or make a new operation
			OUT_Running			:= FALSE;
			OUT_Done			:= FALSE;
			OUT_PositionError	:= FALSE;

			StepTimer.IN	:= TRUE;
			StepTimer.PT	:= t#0.5s;

			IN_SikoData.StartPositioning := FALSE;

			IF StepTimer.Q AND NOT IN_HMI_MoveAt THEN
				IN_SikoData.AbortPositioning := FALSE;
				StepTimer.IN := FALSE;
				Status := 0;
			END_IF

		100:	//Production
			OUT_Running			:= TRUE;
			OUT_Done			:= FALSE;
			OUT_PositionError	:= FALSE;

			OUT_PositionError := FALSE;

			IN_SikoData.StartPositioning := FALSE;

			IF IN_Mode <> 1 THEN
				StepTimer.IN := FALSE;
				Status := 0;
			END_IF

			IF IN_SikoData.MotorDisabled THEN
				StepTimer.IN := FALSE;
				Status := 150;
			END_IF

			IF IN_SikoData.InPosition THEN
				OUT_Done := TRUE;
				StepTimer.IN := FALSE;
				Status := 120;
			ELSE
				IF NOT IN_SikoData.PositioningInProgress AND IN_EnableToRun THEN //v049
					StepTimer.IN := FALSE;
					Status := 110;
				END_IF
			END_IF

		110:	//Production - Wait for positioning
			OUT_Running			:= TRUE;
			OUT_Done			:= FALSE;
			OUT_PositionError	:= FALSE;

			StepTimer.PT	:= t#240s;

			OUT_PositionError := FALSE;

			IN_SikoData.StartPositioning := IN_SikoData.CalibrationDone			AND NOT IN_SikoData.OnError					AND NOT
											IN_SikoData.CommunicationFault		AND NOT IN_SikoData.MotorDisabled			AND IN_SikoData.EmergencyOkFbk	AND NOT
											IN_SikoData.TargetOutsideSwLimit	AND NOT IN_SikoData.DeviceOutsideSwLimit;

			StepTimer.IN := IN_SikoData.StartPositioning;

			//Motor in position
			IF IN_SikoData.InPosition THEN
				StepTimer.IN := FALSE;
				Status := 120;
			END_IF

			IF IN_SikoData.OnError OR StepTimer.Q OR IN_SikoData.CommunicationFault OR IN_SikoData.TargetOutsideSwLimit THEN
				IN_SikoData.AbortPositioning := TRUE;
				IN_SikoData.StartPositioning := FALSE;
				StepTimer.IN := FALSE;
				Status := 130;
			END_IF

			IF NOT IN_SikoData.EmergencyOkFbk THEN
				IN_SikoData.StartPositioning := FALSE;
				StepTimer.IN := FALSE;
				Status := 140;
			END_IF

			IF IN_SikoData.MotorDisabled THEN
				StepTimer.IN := FALSE;
				Status := 150;
			END_IF

			IF IN_Mode <> 1 THEN
				StepTimer.IN := FALSE;
				Status := 190;
			END_IF

		120:	//Motor in position
			OUT_Running			:= TRUE;
			OUT_Done			:= TRUE;
			OUT_PositionError	:= FALSE;

			IN_SikoData.StartPositioning := FALSE;
			StepTimer.IN	:= FALSE;

			IF NOT IN_SikoData.InPosition THEN
				Status := 160;
			END_IF

			IF IN_SikoData.MotorDisabled THEN
				Status := 150;
			END_IF

			IF IN_Mode <> 1 THEN
				Status := 0;
			END_IF

		130:	//Error during positioning phase. Aknoledge required
			OUT_Running			:= TRUE;
			OUT_Done			:= FALSE;
			OUT_PositionError	:= TRUE;

			IN_SikoData.StartPositioning := FALSE;
			StepTimer.IN	:= FALSE;

			IF IN_Reset THEN
				IN_SikoData.AbortPositioning := FALSE;
				OUT_PositionError := FALSE;
				Status := 100;
			END_IF

			IF IN_HMI_MoveAt THEN
				IN_SikoData.AbortPositioning := FALSE;
				OUT_PositionError := FALSE;
				Status := 131;
			END_IF

			IF IN_SikoData.MotorDisabled THEN
				IN_SikoData.AbortPositioning := FALSE;
				OUT_PositionError := FALSE;
				Status := 150;
			END_IF

			IF IN_Mode <> 1 THEN
				IN_SikoData.AbortPositioning :=FALSE;
				StepTimer.PT :=FALSE;
				Status :=0;
			END_IF

		131: 	//Error during positioning phase. Manual positioning
			OUT_Running			:= TRUE;
			OUT_Done			:= FALSE;
			OUT_PositionError	:= FALSE;

			IN_SikoData.StartPositioning := FALSE;
			StepTimer.IN	:= TRUE;
			StepTimer.PT	:= t#240s;

			IN_SikoData.StartPositioning := IN_SikoData.CalibrationDone			AND NOT IN_SikoData.OnError					AND NOT
											IN_SikoData.CommunicationFault		AND NOT IN_SikoData.MotorDisabled			AND IN_SikoData.EmergencyOkFbk	AND NOT
											IN_SikoData.TargetOutsideSwLimit	AND NOT IN_SikoData.DeviceOutsideSwLimit;

			//Motor in position
			IF IN_SikoData.InPosition AND NOT IN_HMI_MoveAt THEN
				IN_SikoData.StartPositioning := FALSE;
				StepTimer.IN := FALSE;
				Status := 120;
			END_IF

			//Timeout positioning
			IF StepTimer.Q THEN
				IN_SikoData.StartPositioning := FALSE;
				IN_SikoData.AbortPositioning := TRUE;
				StepTimer.IN := FALSE;
				Status := 130;
			END_IF

			IF IN_SikoData.MotorDisabled THEN
				IN_SikoData.AbortPositioning := TRUE;
				OUT_PositionError := FALSE;
				Status := 150;
			END_IF

			IF IN_Mode <> 1 THEN
				IN_SikoData.StartPositioning := FALSE;
				IN_SikoData.AbortPositioning := TRUE;
				StepTimer.IN := FALSE;
				Status := 132;
			END_IF

		132:		//Abort command. Wait 0.5s before changing mode or make a new operation
			OUT_Running			:= TRUE;
			OUT_Done			:= FALSE;
			OUT_PositionError	:= FALSE;

			StepTimer.IN	:= TRUE;
			StepTimer.PT	:= t#0.5s;

			IN_SikoData.StartPositioning := FALSE;

			IF StepTimer.Q AND NOT IN_HMI_MoveAt THEN
				IN_SikoData.AbortPositioning := FALSE;
				StepTimer.IN := FALSE;
				Status := 0;
			END_IF

		140:	//Emergency
			OUT_Running			:= TRUE;
			OUT_Done			:= FALSE;
			OUT_PositionError	:= FALSE;

			IN_SikoData.StartPositioning := FALSE;

			IF IN_SikoData.EmergencyOkFbk THEN
				StepTimer.IN := FALSE;
				Status := 100;
			END_IF

			IF IN_SikoData.MotorDisabled THEN
				Status := 150;
			END_IF

			IF IN_Mode <> 1 THEN
				Status := 0;
			END_IF

		150:	//Motor disabled
			OUT_Running			:= TRUE;
			OUT_Done			:= FALSE;
			OUT_PositionError	:= FALSE;

			IN_SikoData.StartPositioning := FALSE;
			IN_SikoData.AbortPositioning := FALSE;

			IF NOT IN_SikoData.MotorDisabled THEN
				StepTimer.IN := FALSE;
				Status := 130;
			END_IF

			IF IN_Mode <> 1 THEN
				Status := 0;
			END_IF

		160:	//Positioning lost
			OUT_Running			:= TRUE;
			OUT_Done			:= FALSE;
			OUT_PositionError	:= FALSE;

			IF IN_SikoData.MotorDisabled OR IN_Reset THEN
				StepTimer.IN := FALSE;
				Status := 100;
			END_IF

			IF IN_Mode <> 1 THEN
				Status := 0;
			END_IF

		190: //Exit step
			OUT_Running			:= FALSE;
			OUT_Done			:= FALSE;
			OUT_PositionError	:= FALSE;

			StepTimer.IN := TRUE;
			StepTimer.PT := t#2s;

			IN_SikoData.AbortPositioning := TRUE;
			IN_SikoData.StartPositioning := FALSE;

			IF StepTimer.Q AND NOT IN_HMI_MoveAt THEN
				IN_SikoData.AbortPositioning := FALSE;
				StepTimer.IN := FALSE;
				Status	:= 0;
			END_IF

		200:	//Cleaning
			OUT_Running			:= TRUE;
			OUT_Done			:= FALSE;
			OUT_PositionError	:= FALSE;

			IN_SikoData.StartPositioning := FALSE;

			IF IN_Mode <> 2 THEN
				StepTimer.IN := FALSE;
				Status := 0;
			END_IF

			IF IN_SikoData.MotorDisabled THEN
				StepTimer.IN := FALSE;
				Status := 250;
			END_IF

			IF IN_SikoData.InPosition THEN
				OUT_Done := TRUE;
				StepTimer.IN := FALSE;
				Status := 220;
			ELSE
				IF NOT IN_SikoData.PositioningInProgress AND IN_EnableToRun THEN //v049
					StepTimer.IN := FALSE;
					Status := 210;
				END_IF
			END_IF

		210:	//Cleaning - Wait for position
			OUT_Running			:= TRUE;
			OUT_Done			:= FALSE;
			OUT_PositionError	:= FALSE;

			StepTimer.PT := t#240s;

			IN_SikoData.StartPositioning := IN_SikoData.CalibrationDone			AND NOT IN_SikoData.OnError					AND NOT
											IN_SikoData.CommunicationFault		AND NOT IN_SikoData.MotorDisabled			AND IN_SikoData.EmergencyOkFbk	AND NOT
											IN_SikoData.TargetOutsideSwLimit	AND NOT IN_SikoData.DeviceOutsideSwLimit;

			StepTimer.IN := IN_SikoData.StartPositioning;

			IF IN_SikoData.InPosition THEN
				StepTimer.IN := FALSE;
				Status := 220;
			END_IF

			IF IN_SikoData.OnError OR StepTimer.Q OR IN_SikoData.CommunicationFault OR IN_SikoData.TargetOutsideSwLimit THEN
				IN_SikoData.AbortPositioning := TRUE;
				IN_SikoData.StartPositioning := FALSE;
				StepTimer.IN := FALSE;
				Status := 230;
			END_IF

			IF NOT IN_SikoData.EmergencyOkFbk THEN
				IN_SikoData.StartPositioning := FALSE;
				StepTimer.IN := FALSE;
				Status := 240;
			END_IF

			IF IN_SikoData.MotorDisabled THEN
				StepTimer.IN := FALSE;
				Status := 250;
			END_IF

			IF IN_Mode <> 2 THEN
				StepTimer.IN := FALSE;
				Status := 290;
			END_IF

		220: 	//Motor in position
			OUT_Running			:= TRUE;
			OUT_Done			:= TRUE;
			OUT_PositionError	:= FALSE;

			IN_SikoData.StartPositioning := FALSE;
			StepTimer.IN := FALSE;

			IF NOT IN_SikoData.InPosition THEN
				Status := 260;
			END_IF

			IF IN_SikoData.MotorDisabled THEN
				Status := 250;
			END_IF

			IF IN_Mode <> 2 THEN
				Status := 0;
			END_IF

		230:
			OUT_Running			:= TRUE;
			OUT_Done			:= FALSE;
			OUT_PositionError	:= TRUE;

			IN_SikoData.StartPositioning := FALSE;
			StepTimer.IN	:= FALSE;

			IF IN_Reset THEN
				IN_SikoData.AbortPositioning := FALSE;
				OUT_PositionError := FALSE;
				Status := 200;
			END_IF

			IF IN_HMI_MoveAt THEN
				IN_SikoData.AbortPositioning := FALSE;
				OUT_PositionError := FALSE;
				Status := 231;
			END_IF

			IF IN_SikoData.MotorDisabled THEN
				IN_SikoData.AbortPositioning := FALSE;
				OUT_PositionError := FALSE;
				Status := 250;
			END_IF

			IF IN_Mode <> 2 THEN
				IN_SikoData.AbortPositioning :=FALSE;
				StepTimer.PT :=FALSE;
				Status :=0;
			END_IF

		231: 	//Error during positioning phase. Manual positioning
			OUT_Running			:= TRUE;
			OUT_Done			:= FALSE;
			OUT_PositionError	:= FALSE;

			IN_SikoData.StartPositioning := FALSE;
			StepTimer.IN	:= TRUE;
			StepTimer.PT	:= t#240s;

			IN_SikoData.StartPositioning := IN_SikoData.CalibrationDone			AND NOT IN_SikoData.OnError					AND NOT
											IN_SikoData.CommunicationFault		AND NOT IN_SikoData.MotorDisabled			AND IN_SikoData.EmergencyOkFbk	AND NOT
											IN_SikoData.TargetOutsideSwLimit	AND NOT IN_SikoData.DeviceOutsideSwLimit;

			//Motor in position
			IF IN_SikoData.InPosition AND NOT IN_HMI_MoveAt THEN
				IN_SikoData.StartPositioning := FALSE;
				StepTimer.IN := FALSE;
				Status := 220;
			END_IF

			//Timeout positioning
			IF StepTimer.Q THEN
				IN_SikoData.StartPositioning := FALSE;
				IN_SikoData.AbortPositioning := TRUE;
				StepTimer.IN := FALSE;
				Status := 230;
			END_IF

			IF IN_SikoData.MotorDisabled THEN
				IN_SikoData.AbortPositioning := TRUE;
				OUT_PositionError := FALSE;
				Status := 250;
			END_IF

			IF IN_Mode <> 1 THEN
				IN_SikoData.StartPositioning := FALSE;
				IN_SikoData.AbortPositioning := TRUE;
				StepTimer.IN := FALSE;
				Status := 232;
			END_IF

		232:		//Abort command. Wait 0.5s before changing mode or make a new operation
			OUT_Running			:= TRUE;
			OUT_Done			:= FALSE;
			OUT_PositionError	:= FALSE;

			StepTimer.IN	:= TRUE;
			StepTimer.PT	:= t#0.5s;

			IN_SikoData.StartPositioning := FALSE;

			IF StepTimer.Q AND NOT IN_HMI_MoveAt THEN
				IN_SikoData.AbortPositioning := FALSE;
				StepTimer.IN := FALSE;
				Status := 0;
			END_IF

		240: 	//Emergency
			OUT_Running			:= TRUE;
			OUT_Done			:= FALSE;
			OUT_PositionError	:= FALSE;

			IN_SikoData.StartPositioning := FALSE;

			IF IN_SikoData.EmergencyOkFbk THEN
				StepTimer.IN := FALSE;
				Status := 200;
			END_IF

			IF IN_SikoData.MotorDisabled THEN
				Status := 250;
			END_IF

			IF IN_Mode <> 2 THEN
				Status := 0;
			END_IF

		250:	//Motor disabled
			OUT_Running			:= TRUE;
			OUT_Done			:= FALSE;
			OUT_PositionError	:= FALSE;

			IN_SikoData.StartPositioning := FALSE;
			IN_SikoData.AbortPositioning := FALSE;

			IF NOT IN_SikoData.MotorDisabled THEN
				StepTimer.IN := FALSE;
				Status := 230;
			END_IF

			IF IN_Mode <> 2 THEN
				Status := 0;
			END_IF

		260:	//Positioning lost
			OUT_Running			:= TRUE;
			OUT_Done			:= FALSE;
			OUT_PositionError	:= FALSE;

			IF IN_SikoData.MotorDisabled OR IN_Reset THEN
				StepTimer.IN := FALSE;
				Status := 200;
			END_IF

			IF IN_Mode <> 2 THEN
				Status := 0;
			END_IF

		290: //Exit step.
			OUT_Running			:= FALSE;
			OUT_Done			:= FALSE;
			OUT_PositionError	:= FALSE;

			StepTimer.IN := TRUE;
			StepTimer.PT := t#2s;

			IN_SikoData.AbortPositioning := TRUE;
			IN_SikoData.StartPositioning := FALSE;

			IF StepTimer.Q AND NOT IN_HMI_MoveAt THEN
				IN_SikoData.AbortPositioning := FALSE;
				StepTimer.IN := FALSE;
				Status	:= 0;
			END_IF

		ELSE
			Status := 0;
	END_CASE
END_FUNCTION_BLOCK
```
